	// 左臂电机
	axis_LeftArm_Wrist_MoveAbs									:MC_MoveAbsolute;			//左臂_腕电机MoveAbs功能块	
	axis_LeftArm_Left_MoveAbs									:MC_MoveAbsolute;			//左臂_左电机MoveAbs功能块
	axis_LeftArm_Right_MoveAbs									:MC_MoveAbsolute;			//左臂_右电机MoveAbs功能块
	axis_LeftArm_Lift_MoveAbs									:MC_MoveAbsolute;			//左臂_升电机MoveAbs功能块
	                                                                                                
	// 右臂电机                                                                                         
	axis_RightArm_Wrist_MoveAbs									:MC_MoveAbsolute;			//右臂_腕电机MoveAbs功能块	
	axis_RightArm_Left_MoveAbs									:MC_MoveAbsolute;			//右臂_左电机MoveAbs功能块
	axis_RightArm_Right_MoveAbs									:MC_MoveAbsolute;			//右臂_右电机MoveAbs功能块
	axis_RightArm_Lift_MoveAbs									:MC_MoveAbsolute;			//右臂_升电机MoveAbs功能块
	                                                                                               
	// 小龙门电机                                                                                        
	axis_SmallGate_Left_MoveAbs									:MC_MoveAbsolute;			//小门_左电机MoveAbs功能块
	axis_SmallGate_Right_MoveAbs								:MC_MoveAbsolute;			//小门_右电机MoveAbs功能块
	                                                                                               
	// 大龙门单电机                                                                                       
	axis_BigGate_Left_MoveAbs									:MC_MoveAbsolute;			//大门_左电机MoveAbs功能块
	axis_BigGate_Right_MoveAbs									:MC_MoveAbsolute;			//大门_右电机MoveAbs功能块
	                                                                                               
	// 后龙门单电机                                                                                      
	axis_BackGate_Left_MoveAbs									:MC_MoveAbsolute;			//后门_左电机MoveAbs功能块
	axis_BackGate_Right_MoveAbs									:MC_MoveAbsolute;			//后门_右电机MoveAbs功能块
	
	// 右轮
	axis_RightWheel_Steer_MoveAbs								:MC_MoveAbsolute;
	axis_RightWheel_Walk_MoveAbs								:MC_MoveAbsolute;
	
	// 左轮
	axis_LeftWheel_Steer_MoveAbs								:MC_MoveAbsolute;
	axis_LeftWheel_Walk_MoveAbs									:MC_MoveAbsolute;

(*======================================== 机器人各轴 MC_MoveAbs定义 End =====================================*)



(*====================================== 机器人各轴 MC_MoveVelocity定义 Start ================================*)

	axis_LeftWheel_Walk_MoveVelo								:MC_MoveVelocity;			// 左轮按速度运动
	axis_RightWheel_Walk_MoveVelo								:MC_MoveVelocity;			// 右轮按速度运动
	
(*====================================== 机器人各轴 MC_MoveVelocity定义 Stop ================================*)



(*======================================== 机器人各轴 MC_Stop定义 Start ==================================*)
	
	// 左臂电机
	axis_LeftArm_Wrist_McStop									:MC_Stop;			//左臂_腕电机MC_Stop块	
	axis_LeftArm_Left_McStop									:MC_Stop;			//左臂_左电机MC_Stop块
	axis_LeftArm_Right_McStop									:MC_Stop;			//左臂_右电机MC_Stop块
	axis_LeftArm_Lift_McStop									:MC_Stop;			//左臂_升电机MC_Stop块
	                                                                                        
	// 右臂电机                                                                                 
	axis_RightArm_Wrist_McStop									:MC_Stop;			//右臂_腕电机MC_Stop块	
	axis_RightArm_Left_McStop									:MC_Stop;			//右臂_左电机MC_Stop块
	axis_RightArm_Right_McStop									:MC_Stop;			//右臂_右电机MC_Stop块
	axis_RightArm_Lift_McStop									:MC_Stop;			//右臂_升电机MC_Stop块
	                                                                                        
	// 小龙门电机                                                                                
	axis_SmallGate_Left_McStop									:MC_Stop;			//小门_左电机MC_Stop块
	axis_SmallGate_Right_McStop									:MC_Stop;			//小门_右电机MC_Stop块
	                                                                                        
	// 大龙门单电机                                                                               
	axis_BigGate_Left_McStop									:MC_Stop;			//大门_左电机MC_Stop块
	axis_BigGate_Right_McStop									:MC_Stop;			//大门_右电机MC_Stop块
	                                                                                        
	// 后龙门单电机                                                                               
	axis_BackGate_Left_McStop									:MC_Stop;			//后门_左电机MC_Stop块
	axis_BackGate_Right_McStop									:MC_Stop;			//后门_右电机MC_Stop块

	// 右轮
	axis_RightWheel_Steer_McStop								:MC_Stop;;
	axis_RightWheel_Walk_McStop									:MC_Stop;
	
	// 左轮
	axis_LeftWheel_Steer_McStop									:MC_Stop;
	axis_LeftWheel_Walk_McStop									:MC_Stop;	
	

(*======================================== 机器人各轴 Mc_Stop定义 End =====================================*)




	

END_VAR

// ---- GVLs/Robot_Parameter.TcGVL
//{attribute 'qualified_only'}
VAR_GLOBAL
	
(* 测试臂参数
	
	//已知量
	h 						:LREAL:=260;
	i 						:LREAL:=260;
	g 						:LREAL:=150;
	f 						:LREAL:=150;
	w 						:LREAL:=110;
	angle_a					:LREAL:=137.5;			// 单位为度
	j						:LREAL:=40;
	n						:LREAL:=290.7497;     	// 余弦定理
	angle_FCE				:LREAL:=5.3330;			//余弦定理（单位为度）
*)

	// Left arm parameter
	LeftArm_h				:LREAL:=584.21;
	LeftArm_i				:LREAL:=500;
	LeftArm_g				:LREAL:=418;
	LeftArm_f				:LREAL:=418;
	LeftArm_w				:LREAL:=110;
	LeftArm_angle_a			:LREAL:=134.7;			//数模实测值,单位为度
	LeftArm_j				:LREAL:=147.73;
	LeftArm_n				:LREAL:=612.98;			//数模实测值
	LeftArm_angle_FCE		:LREAL:=9.86;			//数模实测值,单位为度
	
	// Right arm parameter
	RightArm_h				:LREAL:=500;
	RightArm_i				:LREAL:=584.21;
	RightArm_g				:LREAL:=418;
	RightArm_f				:LREAL:=418;
	RightArm_w				:LREAL:=110;
	RightArm_angle_a		:LREAL:=137.57;			//单位度
	RightArm_j				:LREAL:=147.73;
	RightArm_m				:LREAL:=617.76;
	RightArm_angle_FDE		:LREAL:=9.29;			//单位度

	//常量
	PI						:LREAL:=3.1415926;
	

END_VAR

// ---- GVLs/Robot_Status_Info.TcGVL
//{attribute 'qualified_only'}
VAR_GLOBAL
	
	(**********************************   电池相关参数    *************************************)
											
	Battery_TotalVoltage		AT%MW300		:LREAL;			 //voltage, unit: V
	Battery_TotalCurrent		AT%MW304		:LREAL;			 //current, unit:A
	Battery_RemainCapacity						:REAL;			 //remain capacitu, unit:Ah
	Battery_NominalCapacity						:REAL;			 //nominal capacity, unit:Ah
	Battery_CycleNum							:UINT;			 //cycle number, unit:times
	Battery_ProtectionMode						:WORD;			 //protection mode word
	Battery_RSOC								:USINT;			 //remain capacity, unit:%
	Battery_FETStatus							:BYTE;			 //mos fet status word
	Battery_humidity							:USINT;			 //humidity, unity:%
	Battery_WarningStatus						:WORD;			 //warning status word
	
	// 自定义标志位
	bBattery_Charging	   	 	    AT%MX10.0	:BOOL;			 //电池充放电状态标志位，电流正为充电，电流负为放电。
	bBattery_DisCharging		    AT%MX10.1	:BOOL;			 //电池充放电状态标志位，电流正为充电，电流负为放电。
	lrBattery_DisChargingCurrent	AT%MW304	:LREAL;			 //放电电流
	lrBattery_ChargingCurrent		AT%MW308	:LREAL;			 //充电电流
	lrBattery_RemainCapacity_Pecent AT%MW312	:LREAL;			 //剩余电量百分比，和Battery_RSOC不同，这个是用Battery_RemainCapacity、Battery_NominalCapacity两个参数算出来的。
	
	// Battery_ProtectionMode 电池保护状态定义标志位
	bSingleCellOvervoltageProtection    		: BOOL;			 // bit0: 单体过压保护
	bSingleCellUndervoltageProtection   		: BOOL;			 // bit1: 单体欠压保护
	bWholeGroupOvervoltageProtection    		: BOOL;			 // bit2: 整组过压保护
	bWholeGroupUndervoltageProtection   		: BOOL;			 // bit3: 整组欠压保护
	bChargingOverTemperatureProtection  		: BOOL;			 // bit4: 充电过温保护
	bChargingLowTemperatureProtection   		: BOOL;			 // bit5: 充电低温保护
	bDischargingOverTemperatureProtection		: BOOL;			 // bit6: 放电过温保护
	bDischargingLowTemperatureProtection		: BOOL;			 // bit7: 放电低温保护
	bChargingOvercurrentProtection      		: BOOL;			 // bit8: 充电过流保护
	bDischargingOvercurrentProtection   		: BOOL;			 // bit9: 放电过流保护
	bShortCircuitProtection             		: BOOL;			 // bit10: 短路保护
	bFrontEndDetectionICError           		: BOOL;			 // bit11: 前端检测IC错误
	bSoftwareLockedMOS                  		: BOOL;			 // bit12: 软件锁定MOS
	bChargingMOSBreakdownFlag           		: BOOL;			 // bit13: 充电MOS击穿标志
	bDischargingMOSBreakdownFlag        		: BOOL;			 // bit14: 放电MOS击穿标志
	bReserved                           		: BOOL;			 // bit15: 预留

	// Battery_FETStatus 电池MOS标志位
	bChargeMOSStatus    						: BOOL; 		// bit0: 充电MOS状态
	bDischargeMOSStatus 						: BOOL; 		// bit1: 放电MOS状态
	bCurrentLimitStatus 						: BOOL; 		// bit2: 限流模块状态
	bHeatingStatus      						: BOOL; 		// bit3: 加热模块状态
	
	// Battery Warning Status
	bSingleCellHighVoltageWarning    			: BOOL; 		// bit0: 单体高压告警
	bSingleCellLowVoltageWarning     			: BOOL; 		// bit1: 单体低压告警
	bWholeGroupHighVoltageWarning    			: BOOL; 		// bit2: 整组高压告警
	bWholeGroupLowVoltageWarning     			: BOOL; 		// bit3: 整组低压告警
	bChargingHighTemperatureWarning  			: BOOL; 		// bit4: 充电高温告警
	bChargingLowTemperatureWarning   			: BOOL; 		// bit5: 充电低温告警
	bDischargingHighTemperatureWarning			: BOOL; 		// bit6: 放电高温告警
	bDischargingLowTemperatureWarning 			: BOOL; 		// bit7: 放电低温保护
	bChargingHighCurrentWarning      			: BOOL; 		// bit8: 充电电流大告警
	bDischargingHighCurrentWarning   			: BOOL; 		// bit9: 放电电流大告警
	bSingleCellVoltageDifferenceWarning			: BOOL; 		// bit10: 单体压差大告警
	bLowCapacityWarning              			: BOOL; 		// bit11: 容量低告警
	bReserved12                      			: BOOL; 		// bit12: 预留
	bReserved13                      			: BOOL; 		// bit13: 预留
	bReserved14                      			: BOOL; 		// bit14: 预留
	
	
	



	(**********************************   轴相关参数    *************************************)
	
	// 伺服驱动器Error标志位
	bDriverDeviceError_axis_LeftArm_Left				AT%I*					:BOOL;		// 伺服驱动器报警_标志位_LeftArm_Left	
	bDriverDeviceError_axis_LeftArm_Right				AT%I*					:BOOL;		// 伺服驱动器报警_标志位_LeftArm_Right	
	bDriverDeviceError_axis_LeftArm_Wrist				AT%I*					:BOOL;		// 伺服驱动器报警_标志位_LeftArm_Wrist	
	bDriverDeviceError_axis_LeftArm_Lift				AT%I*					:BOOL;		// 伺服驱动器报警_标志位_LeftArm_Lift	
	bDriverDeviceError_axis_RightArm_Left				AT%I*					:BOOL;		// 伺服驱动器报警_标志位_RightArm_Left	
	bDriverDeviceError_axis_RightArm_Right				AT%I*					:BOOL;      // 伺服驱动器报警_标志位_RightArm_Right	
	bDriverDeviceError_axis_RightArm_Wrist				AT%I*					:BOOL;      // 伺服驱动器报警_标志位_RightArm_Wrist	
	bDriverDeviceError_axis_RightArm_Lift				AT%I*					:BOOL;	    // 伺服驱动器报警_标志位_RightArm_Lift	
	bDriverDeviceError_axis_BigGate_Left				AT%I*					:BOOL;		// 伺服驱动器报警_标志位_BigGate_Left
	bDriverDeviceError_axis_BigGate_Right				AT%I*					:BOOL;      // 伺服驱动器报警_标志位_BigGate_Right
	bDriverDeviceError_axis_SmallGate_Left				AT%I*					:BOOL;      // 伺服驱动器报警_标志位_SmallGate_Left
	bDriverDeviceError_axis_SmallGate_Right				AT%I*					:BOOL;      // 伺服驱动器报警_标志位_SmallGate_Right
	bDriverDeviceError_axis_BackGate_Left				AT%I*					:BOOL;		// 伺服驱动器报警_标志位_BackGate_Left
	bDriverDeviceError_axis_BackGate_Right				AT%I*					:BOOL;	    // 伺服驱动器报警_标志位_BackGate_Right
	bDriverDeviceError_axis_RightWheel_Steer			AT%I*					:BOOL;      // 伺服驱动器报警_标志位_RightWheel_Steer
	bDriverDeviceError_axis_RightWheel_Walk				AT%I*					:BOOL;		// 伺服驱动器报警_标志位_RightWheel_Walk
	bDriverDeviceError_axis_LeftWheel_Steer				AT%I*					:BOOL;		// 伺服驱动器报警_标志位_LeftWheel_Steer
	bDriverDeviceError_axis_LeftWheel_Walk				AT%I*					:BOOL;		// 伺服驱动器报警_标志位_LeftWheel_Walk
	
	// 伺服驱动器ErrorCode
	bDriverDeviceErrorCode_axis_LeftArm_Left			AT%I*					:UDINT;		// 伺服驱动器报警_错误代码_LeftArm_Left	
	bDriverDeviceErrorCode_axis_LeftArm_Right			AT%I*					:UDINT;		// 伺服驱动器报警_错误代码_LeftArm_Right	
	bDriverDeviceErrorCode_axis_LeftArm_Wrist			AT%I*					:UDINT;		// 伺服驱动器报警_错误代码_LeftArm_Wrist	
	bDriverDeviceErrorCode_axis_LeftArm_Lift			AT%I*					:UDINT;		// 伺服驱动器报警_错误代码_LeftArm_Lift	
	bDriverDeviceErrorCode_axis_RightArm_Left			AT%I*					:UDINT;		// 伺服驱动器报警_错误代码_RightArm_Left	
	bDriverDeviceErrorCode_axis_RightArm_Right			AT%I*					:UDINT;      // 伺服驱动器报警_错误代码_RightArm_Right	
	bDriverDeviceErrorCode_axis_RightArm_Wrist			AT%I*					:UDINT;      // 伺服驱动器报警_错误代码_RightArm_Wrist	
	bDriverDeviceErrorCode_axis_RightArm_Lift			AT%I*					:UDINT;	    // 伺服驱动器报警_错误代码_RightArm_Lift	
	bDriverDeviceErrorCode_axis_BigGate_Left			AT%I*					:UDINT;		// 伺服驱动器报警_错误代码_BigGate_Left
	bDriverDeviceErrorCode_axis_BigGate_Right			AT%I*					:UDINT;      // 伺服驱动器报警_错误代码_BigGate_Right
	bDriverDeviceErrorCode_axis_SmallGate_Left			AT%I*					:UDINT;      // 伺服驱动器报警_错误代码_SmallGate_Left
	bDriverDeviceErrorCode_axis_SmallGate_Right			AT%I*					:UDINT;      // 伺服驱动器报警_错误代码_SmallGate_Right
	bDriverDeviceErrorCode_axis_BackGate_Left			AT%I*					:UDINT;		// 伺服驱动器报警_错误代码_BackGate_Left
	bDriverDeviceErrorCode_axis_BackGate_Right			AT%I*					:UDINT;	    // 伺服驱动器报警_错误代码_BackGate_Right
	bDriverDeviceErrorCode_axis_RightWheel_Steer		AT%I*					:UDINT;      // 伺服驱动器报警_错误代码_RightWheel_Steer
	bDriverDeviceErrorCode_axis_RightWheel_Walk			AT%I*					:UDINT;		// 伺服驱动器报警_错误代码_RightWheel_Walk
	bDriverDeviceErrorCode_axis_LeftWheel_Steer			AT%I*					:UDINT;		// 伺服驱动器报警_错误代码_LeftWheel_Steer
	bDriverDeviceErrorCode_axis_LeftWheel_Walk			AT%I*					:UDINT;		// 伺服驱动器报警_错误代码_LeftWheel_Walk
	
END_VAR

// ---- POUs/AxisAbs.TcPOU
PROGRAM AxisAbs
VAR
	nSpeed_MoveAbs						:LREAL:=5;
	
	nTargetPos_MoveAbs								:LREAL;

END_VAR


// LeftArm_Left_MoveAbs
IF bManualCtrl_Part_LeftArm_Left THEN					
	axis_LeftArm_Left_MoveAbs(
		Axis:= axis_LeftArm_Left, 
		Execute:= bAxis_LeftArm_Left_MoveAbs, 
		Position:= nTargetPos_MoveAbs, 
		Velocity:= nSpeed_MoveAbs, 
		Acceleration:= , 
		Deceleration:= , 
		Jerk:= , 
		BufferMode:= , 
		Options:= , 
		Done=> , 
		Busy=> , 
		Active=> , 
		CommandAborted=> , 
		Error=> , 
		ErrorID=> );	
END_IF

// LeftArm_Right_MoveAbs
IF bManualCtrl_Part_LeftArm_Right THEN					
	axis_LeftArm_Right_MoveAbs(
		Axis:= axis_LeftArm_Right, 
		Execute:= bAxis_LeftArm_Right_MoveAbs, 
		Position:= nTargetPos_MoveAbs, 
		Velocity:= nSpeed_MoveAbs, 
		Acceleration:= , 
		Deceleration:= , 
		Jerk:= , 
		BufferMode:= , 
		Options:= , 
		Done=> , 
		Busy=> , 
		Active=> , 
		CommandAborted=> , 
		Error=> , 
		ErrorID=> );	
END_IF


// LeftArm_Wrist_MoveAbs
IF bManualCtrl_Part_LeftArm_Wrist THEN					
	axis_LeftArm_Wrist_MoveAbs(
		Axis:= axis_LeftArm_Wrist, 
		Execute:= bAxis_LeftArm_Wrist_MoveAbs, 
		Position:= nTargetPos_MoveAbs, 
		Velocity:= nSpeed_MoveAbs, 
		Acceleration:= , 
		Deceleration:= , 
		Jerk:= , 
		BufferMode:= , 
		Options:= , 
		Done=> , 
		Busy=> , 
		Active=> , 
		CommandAborted=> , 
		Error=> , 
		ErrorID=> );	
END_IF


// LeftArm_Lift_MoveAbs
IF bManualCtrl_Part_LeftArm_Lift THEN					
	axis_LeftArm_Lift_MoveAbs(
		Axis:= axis_LeftArm_Lift, 
		Execute:= bAxis_LeftArm_Lift_MoveAbs, 
		Position:= nTargetPos_MoveAbs, 
		Velocity:= nSpeed_MoveAbs, 
		Acceleration:= , 
		Deceleration:= , 
		Jerk:= , 
		BufferMode:= , 
		Options:= , 
		Done=> , 
		Busy=> , 
		Active=> , 
		CommandAborted=> , 
		Error=> , 
		ErrorID=> );	
END_IF



// RightArm_Left_MoveAbs
IF bManualCtrl_Part_RightArm_Left THEN					
	axis_RightArm_Left_MoveAbs(
		Axis:= axis_RightArm_Left, 
		Execute:= bAxis_RightArm_Left_MoveAbs, 
		Position:= nTargetPos_MoveAbs, 
		Velocity:= nSpeed_MoveAbs, 
		Acceleration:= , 
		Deceleration:= , 
		Jerk:= , 
		BufferMode:= , 
		Options:= , 
		Done=> , 
		Busy=> , 
		Active=> , 
		CommandAborted=> , 
		Error=> , 
		ErrorID=> );	
END_IF

// RightArm_Right_MoveAbs
IF bManualCtrl_Part_RightArm_Right THEN					
	axis_RightArm_Right_MoveAbs(
		Axis:= axis_RightArm_Right, 
		Execute:= bAxis_RightArm_Right_MoveAbs, 
		Position:= nTargetPos_MoveAbs, 
		Velocity:= nSpeed_MoveAbs, 
		Acceleration:= , 
		Deceleration:= , 
		Jerk:= , 
		BufferMode:= , 
		Options:= , 
		Done=> , 
		Busy=> , 
		Active=> , 
		CommandAborted=> , 
		Error=> , 
		ErrorID=> );	
END_IF


// RightArm_Wrist_MoveAbs
IF bManualCtrl_Part_RightArm_Wrist THEN					
	axis_RightArm_Wrist_MoveAbs(
		Axis:= axis_RightArm_Wrist, 
		Execute:= bAxis_RightArm_Wrist_MoveAbs, 
		Position:= nTargetPos_MoveAbs, 
		Velocity:= nSpeed_MoveAbs, 
		Acceleration:= , 
		Deceleration:= , 
		Jerk:= , 
		BufferMode:= , 
		Options:= , 
		Done=> , 
		Busy=> , 
		Active=> , 
		CommandAborted=> , 
		Error=> , 
		ErrorID=> );	
END_IF


// RightArm_Lift_MoveAbs
IF bManualCtrl_Part_RightArm_Lift THEN					
	axis_RightArm_Lift_MoveAbs(
		Axis:= axis_RightArm_Lift, 
		Execute:= bAxis_RightArm_Lift_MoveAbs, 
		Position:= nTargetPos_MoveAbs, 
		Velocity:= nSpeed_MoveAbs, 
		Acceleration:= , 
		Deceleration:= , 
		Jerk:= , 
		BufferMode:= , 
		Options:= , 
		Done=> , 
		Busy=> , 
		Active=> , 
		CommandAborted=> , 
		Error=> , 
		ErrorID=> );	
END_IF


// BigGate_Left_MoveAbs
IF bManualCtrl_Part_BigGate_Left THEN					
	axis_BigGate_Left_MoveAbs(
		Axis:= axis_BigGate_Left, 
		Execute:= bAxis_BigGate_Left_MoveAbs, 
		Position:= nTargetPos_MoveAbs, 
		Velocity:= nSpeed_MoveAbs, 
		Acceleration:= , 
		Deceleration:= , 
		Jerk:= , 
		BufferMode:= , 
		Options:= , 
		Done=> , 
		Busy=> , 
		Active=> , 
		CommandAborted=> , 
		Error=> , 
		ErrorID=> );	
END_IF

// BigGate_Right_MoveAbs
IF bManualCtrl_Part_BigGate_Right THEN					
	axis_BigGate_Right_MoveAbs(
		Axis:= axis_BigGate_Right, 
		Execute:= bAxis_BigGate_Right_MoveAbs, 
		Position:= nTargetPos_MoveAbs, 
		Velocity:= nSpeed_MoveAbs, 
		Acceleration:= , 
		Deceleration:= , 
		Jerk:= , 
		BufferMode:= , 
		Options:= , 
		Done=> , 
		Busy=> , 
		Active=> , 
		CommandAborted=> , 
		Error=> , 
		ErrorID=> );	
END_IF

// SmallGate_Left_MoveAbs
IF bManualCtrl_Part_SmallGate_Left THEN					
	axis_SmallGate_Left_MoveAbs(
		Axis:= axis_SmallGate_Left, 
		Execute:= bAxis_SmallGate_Left_MoveAbs, 
		Position:= nTargetPos_MoveAbs, 
		Velocity:= nSpeed_MoveAbs, 
		Acceleration:= , 
		Deceleration:= , 
		Jerk:= , 
		BufferMode:= , 
		Options:= , 
		Done=> , 
		Busy=> , 
		Active=> , 
		CommandAborted=> , 
		Error=> , 
		ErrorID=> );	
END_IF

// SmallGate_Right_MoveAbs
IF bManualCtrl_Part_SmallGate_Right THEN					
	axis_SmallGate_Right_MoveAbs(
		Axis:= axis_SmallGate_Right, 
		Execute:= bAxis_SmallGate_Right_MoveAbs, 
		Position:= nTargetPos_MoveAbs, 
		Velocity:= nSpeed_MoveAbs, 
		Acceleration:= , 
		Deceleration:= , 
		Jerk:= , 
		BufferMode:= , 
		Options:= , 
		Done=> , 
		Busy=> , 
		Active=> , 
		CommandAborted=> , 
		Error=> , 
		ErrorID=> );	
END_IF


// BackGate_Left_MoveAbs
IF bManualCtrl_Part_BackGate_Left THEN					
	axis_BackGate_Left_MoveAbs(
		Axis:= axis_BackGate_Left, 
		Execute:= bAxis_BackGate_Left_MoveAbs, 
		Position:= nTargetPos_MoveAbs, 
		Velocity:= nSpeed_MoveAbs, 
		Acceleration:= , 
		Deceleration:= , 
		Jerk:= , 
		BufferMode:= , 
		Options:= , 
		Done=> , 
		Busy=> , 
		Active=> , 
		CommandAborted=> , 
		Error=> , 
		ErrorID=> );	
END_IF

// BackGate_Right_MoveAbs
IF bManualCtrl_Part_BackGate_Right THEN					
	axis_BackGate_Right_MoveAbs(
		Axis:= axis_BackGate_Right, 
		Execute:= bAxis_BackGate_Right_MoveAbs, 
		Position:= nTargetPos_MoveAbs, 
		Velocity:= nSpeed_MoveAbs, 
		Acceleration:= , 
		Deceleration:= , 
		Jerk:= , 
		BufferMode:= , 
		Options:= , 
		Done=> , 
		Busy=> , 
		Active=> , 
		CommandAborted=> , 
		Error=> , 
		ErrorID=> );	
END_IF

END_PROGRAM

// ---- POUs/AxisAllCtrl.TcPOU
PROGRAM AxisAllCtrl
VAR
	i				:USINT := 1;

END_VAR



//所有Axis上电
IF bAxis_All_Enable THEN
	FOR i:=1 TO nAxisNum DO
		aAxis_All_Enable_Group[i]^:=TRUE;
	END_FOR
END_IF

//所有Axis下电
IF bAxis_All_Disable THEN
	FOR i:=1 TO nAxisNum DO
		aAxis_All_Enable_Group[i]^:=FALSE;
	END_FOR
END_IF

//所有轴清除故障
IF bAxis_All_Reset THEN
	FOR i:=1 TO nAxisNum DO
		aAxis_All_Reset_Group[i]^:=TRUE;
	END_FOR
ELSE
	FOR i:=1 TO nAxisNum DO
		aAxis_All_Reset_Group[i]^:=FALSE;
	END_FOR	
END_IF

END_PROGRAM

// ---- POUs/AxisJog.TcPOU
PROGRAM AxisJog
VAR
	lrJogSpeed	: POINTER TO LREAL;
END_VAR

// 快速Jog速度设定
IF bJogFast THEN
	lrJogSpeed := ADR(aAxis_Jog_Speed[1]);
ELSE
	lrJogSpeed := ADR(aAxis_Jog_Speed[0]);
END_IF

// LeftArm_Left_Jog
IF bManualCtrl_Part_LeftArm_Left THEN

	axis_LeftArm_Left_Jog(
		Axis:= axis_LeftArm_Left, 
		JogForward:= bAxis_LeftArm_Left_JogP , 			// 如果想ABS的时候按下JOG按键不停止ABS动作就加上后面的判断AND NOT axis_LeftArm_Left_MoveAbs.Active
		JogBackwards:= bAxis_LeftArm_Left_JogN, 		// 如果想ABS的时候按下JOG按键不停止ABS动作就加上后面的判断AND NOT axis_LeftArm_Left_MoveAbs.Active
		Mode:= MC_JOGMODE_CONTINOUS, 					//需要设置为MC_JOGMODE_CONTINOUS下面的速度设定才有效
		Position:= , 
		Velocity:= lrJogSpeed^, 
		Acceleration:= , 
		Deceleration:= , 
		Jerk:= , 
		Done=> , 
		Busy=> , 
		Active=> , 
		CommandAborted=> , 
		Error=> , 
		ErrorID=> );

END_IF

// LeftArm_Right_Jog
IF bManualCtrl_Part_LeftArm_Right THEN

	axis_LeftArm_Right_Jog(
		Axis:= axis_LeftArm_Right, 
		JogForward:= bAxis_LeftArm_Right_JogP , 			
		JogBackwards:= bAxis_LeftArm_Right_JogN, 		
		Mode:= MC_JOGMODE_CONTINOUS, 					//需要设置为MC_JOGMODE_CONTINOUS下面的速度设定才有效
		Position:= , 
		Velocity:= lrJogSpeed^, 
		Acceleration:= , 
		Deceleration:= , 
		Jerk:= , 
		Done=> , 
		Busy=> , 
		Active=> , 
		CommandAborted=> , 
		Error=> , 
		ErrorID=> );

END_IF

// LeftArm_Wrist_Jog
IF bManualCtrl_Part_LeftArm_Wrist THEN

	axis_LeftArm_Right_Jog(
		Axis:= axis_LeftArm_Wrist, 
		JogForward:= bAxis_LeftArm_Wrist_JogP , 			
		JogBackwards:= bAxis_LeftArm_Wrist_JogN, 		
		Mode:= MC_JOGMODE_CONTINOUS, 					//需要设置为MC_JOGMODE_CONTINOUS下面的速度设定才有效
		Position:= , 
		Velocity:= lrJogSpeed^, 
		Acceleration:= , 
		Deceleration:= , 
		Jerk:= , 
		Done=> , 
		Busy=> , 
		Active=> , 
		CommandAborted=> , 
		Error=> , 
		ErrorID=> );

END_IF


// LeftArm_Lift_Jog
IF bManualCtrl_Part_LeftArm_Lift THEN

	axis_LeftArm_Lift_Jog(
		Axis:= axis_LeftArm_Lift, 
		JogForward:= bAxis_LeftArm_Lift_JogP , 			
		JogBackwards:= bAxis_LeftArm_Lift_JogN, 		
		Mode:= MC_JOGMODE_CONTINOUS, 					//需要设置为MC_JOGMODE_CONTINOUS下面的速度设定才有效
		Position:= , 
		Velocity:= lrJogSpeed^, 
		Acceleration:= , 
		Deceleration:= , 
		Jerk:= , 
		Done=> , 
		Busy=> , 
		Active=> , 
		CommandAborted=> , 
		Error=> , 
		ErrorID=> );

END_IF



// RightArm_Left_Jog
IF bManualCtrl_Part_RightArm_Left THEN

	axis_RightArm_Left_Jog(
		Axis:= axis_RightArm_Left, 
		JogForward:= bAxis_RightArm_Left_JogP , 			// 如果想ABS的时候按下JOG按键不停止ABS动作就加上后面的判断AND NOT axis_LeftArm_Left_MoveAbs.Active
		JogBackwards:= bAxis_RightArm_Left_JogN, 		// 如果想ABS的时候按下JOG按键不停止ABS动作就加上后面的判断AND NOT axis_LeftArm_Left_MoveAbs.Active
		Mode:= MC_JOGMODE_CONTINOUS, 					//需要设置为MC_JOGMODE_CONTINOUS下面的速度设定才有效
		Position:= , 
		Velocity:= lrJogSpeed^, 
		Acceleration:= , 
		Deceleration:= , 
		Jerk:= , 
		Done=> , 
		Busy=> , 
		Active=> , 
		CommandAborted=> , 
		Error=> , 
		ErrorID=> );

END_IF

// RightArm_Right_Jog
IF bManualCtrl_Part_RightArm_Right THEN

	axis_RightArm_Right_Jog(
		Axis:= axis_RightArm_Right, 
		JogForward:= bAxis_RightArm_Right_JogP , 			
		JogBackwards:= bAxis_RightArm_Right_JogN, 		
		Mode:= MC_JOGMODE_CONTINOUS, 					//需要设置为MC_JOGMODE_CONTINOUS下面的速度设定才有效
		Position:= , 
		Velocity:= lrJogSpeed^, 
		Acceleration:= , 
		Deceleration:= , 
		Jerk:= , 
		Done=> , 
		Busy=> , 
		Active=> , 
		CommandAborted=> , 
		Error=> , 
		ErrorID=> );

END_IF

// RightArm_Wrist_Jog
IF bManualCtrl_Part_RightArm_Wrist THEN

	axis_RightArm_Right_Jog(
		Axis:= axis_RightArm_Wrist, 
		JogForward:= bAxis_RightArm_Wrist_JogP , 			
		JogBackwards:= bAxis_RightArm_Wrist_JogN, 		
		Mode:= MC_JOGMODE_CONTINOUS, 					//需要设置为MC_JOGMODE_CONTINOUS下面的速度设定才有效
		Position:= , 
		Velocity:= lrJogSpeed^, 
		Acceleration:= , 
		Deceleration:= , 
		Jerk:= , 
		Done=> , 
		Busy=> , 
		Active=> , 
		CommandAborted=> , 
		Error=> , 
		ErrorID=> );

END_IF


// RightArm_Lift_Jog
IF bManualCtrl_Part_RightArm_Lift THEN

	axis_RightArm_Lift_Jog(
		Axis:= axis_RightArm_Lift, 
		JogForward:= bAxis_RightArm_Lift_JogP , 			
		JogBackwards:= bAxis_RightArm_Lift_JogN, 		
		Mode:= MC_JOGMODE_CONTINOUS, 					//需要设置为MC_JOGMODE_CONTINOUS下面的速度设定才有效
		Position:= , 
		Velocity:= lrJogSpeed^, 
		Acceleration:= , 
		Deceleration:= , 
		Jerk:= , 
		Done=> , 
		Busy=> , 
		Active=> , 
		CommandAborted=> , 
		Error=> , 
		ErrorID=> );

END_IF


// BigGate_Left_Jog(正转升，反转降)
IF bManualCtrl_Part_BigGate_Left THEN

	axis_BigGate_Left_Jog(
		Axis:= axis_BigGate_Left, 
		JogForward:= bAxis_BigGate_Left_JogP , 			// 如果想ABS的时候按下JOG按键不停止ABS动作就加上后面的判断AND NOT axis_LeftArm_Left_MoveAbs.Active
		JogBackwards:= bAxis_BigGate_Left_JogN, 		// 如果想ABS的时候按下JOG按键不停止ABS动作就加上后面的判断AND NOT axis_LeftArm_Left_MoveAbs.Active
		Mode:= MC_JOGMODE_CONTINOUS, 					//需要设置为MC_JOGMODE_CONTINOUS下面的速度设定才有效
		Position:= , 
		Velocity:= lrJogSpeed^, 
		Acceleration:= , 
		Deceleration:= , 
		Jerk:= , 
		Done=> , 
		Busy=> , 
		Active=> , 
		CommandAborted=> , 
		Error=> , 
		ErrorID=> );

END_IF

// BigGate_Right_Jog(正转降反转升)
IF bManualCtrl_Part_BigGate_Right THEN

	axis_BigGate_Right_Jog(
		Axis:= axis_BigGate_Right, 
		JogForward:= bAxis_BigGate_Right_JogP , 			
		JogBackwards:= bAxis_BigGate_Right_JogN, 		
		Mode:= MC_JOGMODE_CONTINOUS, 					//需要设置为MC_JOGMODE_CONTINOUS下面的速度设定才有效
		Position:= , 
		Velocity:= lrJogSpeed^, 
		Acceleration:= , 
		Deceleration:= , 
		Jerk:= , 
		Done=> , 
		Busy=> , 
		Active=> , 
		CommandAborted=> , 
		Error=> , 
		ErrorID=> );

END_IF


// SmallGate_Left_Jog
IF bManualCtrl_Part_SmallGate_Left THEN

	axis_SmallGate_Left_Jog(
		Axis:= axis_SmallGate_Left, 
		JogForward:= bAxis_SmallGate_Left_JogP , 			// 如果想ABS的时候按下JOG按键不停止ABS动作就加上后面的判断AND NOT axis_LeftArm_Left_MoveAbs.Active
		JogBackwards:= bAxis_SmallGate_Left_JogN, 		// 如果想ABS的时候按下JOG按键不停止ABS动作就加上后面的判断AND NOT axis_LeftArm_Left_MoveAbs.Active
		Mode:= MC_JOGMODE_CONTINOUS, 					//需要设置为MC_JOGMODE_CONTINOUS下面的速度设定才有效
		Position:= , 
		Velocity:= lrJogSpeed^, 
		Acceleration:= , 
		Deceleration:= , 
		Jerk:= , 
		Done=> , 
		Busy=> , 
		Active=> , 
		CommandAborted=> , 
		Error=> , 
		ErrorID=> );

END_IF

// SmallGate_Right_Jog
IF bManualCtrl_Part_SmallGate_Right THEN

	axis_SmallGate_Right_Jog(
		Axis:= axis_SmallGate_Right, 
		JogForward:= bAxis_SmallGate_Right_JogP , 			
		JogBackwards:= bAxis_SmallGate_Right_JogN, 		
		Mode:= MC_JOGMODE_CONTINOUS, 					//需要设置为MC_JOGMODE_CONTINOUS下面的速度设定才有效
		Position:= , 
		Velocity:= lrJogSpeed^, 
		Acceleration:= , 
		Deceleration:= , 
		Jerk:= , 
		Done=> , 
		Busy=> , 
		Active=> , 
		CommandAborted=> , 
		Error=> , 
		ErrorID=> );

END_IF



// BackGate_Left_Jog
IF bManualCtrl_Part_BackGate_Left THEN

	axis_BackGate_Left_Jog(
		Axis:= axis_BackGate_Left, 
		JogForward:= bAxis_BackGate_Left_JogP , 			// 如果想ABS的时候按下JOG按键不停止ABS动作就加上后面的判断AND NOT axis_LeftArm_Left_MoveAbs.Active
		JogBackwards:= bAxis_BackGate_Left_JogN, 		// 如果想ABS的时候按下JOG按键不停止ABS动作就加上后面的判断AND NOT axis_LeftArm_Left_MoveAbs.Active
		Mode:= MC_JOGMODE_CONTINOUS, 					//需要设置为MC_JOGMODE_CONTINOUS下面的速度设定才有效
		Position:= , 
		Velocity:= lrJogSpeed^, 
		Acceleration:= , 
		Deceleration:= , 
		Jerk:= , 
		Done=> , 
		Busy=> , 
		Active=> , 
		CommandAborted=> , 
		Error=> , 
		ErrorID=> );

END_IF

// BackGate_Right_Jog
IF bManualCtrl_Part_BackGate_Right THEN

	axis_BackGate_Right_Jog(
		Axis:= axis_BackGate_Right, 
		JogForward:= bAxis_BackGate_Right_JogP , 			
		JogBackwards:= bAxis_BackGate_Right_JogN, 		
		Mode:= MC_JOGMODE_CONTINOUS, 					//需要设置为MC_JOGMODE_CONTINOUS下面的速度设定才有效
		Position:= , 
		Velocity:= lrJogSpeed^, 
		Acceleration:= , 
		Deceleration:= , 
		Jerk:= , 
		Done=> , 
		Busy=> , 
		Active=> , 
		CommandAborted=> , 
		Error=> , 
		ErrorID=> );

END_IF

END_PROGRAM

// ---- POUs/AxisPowerOn.TcPOU
PROGRAM AxisPowerOn
VAR

END_VAR


//左臂-左电机-PowerOn
axis_LeftArm_Left_Power(
	Axis:= axis_LeftArm_Left, 
	Enable:= bAxis_LeftArm_Left_Enable, 
	Enable_Positive:= TRUE, 
	Enable_Negative:= TRUE, 
	Override:= , 
	BufferMode:= , 
	Options:= , 
	Status=> axis_LeftArm_Left_Power_Output.Done, 
	Busy=> , 
	Error=> , 
	ErrorID=> );
	
	
//左臂-右电机-PowerOn
axis_LeftArm_Right_Power(
	Axis:= axis_LeftArm_Right, 
	Enable:= bAxis_LeftArm_Right_Enable, 
	Enable_Positive:= TRUE, 
	Enable_Negative:= TRUE, 
	Override:= , 
	BufferMode:= , 
	Options:= , 
	Status=> axis_LeftArm_Right_Power_Output.Done, 
	Busy=> , 
	Error=> , 
	ErrorID=> );
	
axis_LeftArm_Lift_Power(
	Axis:= axis_LeftArm_Lift, 
	Enable:= bAxis_LeftArm_Lift_Enable, 
	Enable_Positive:= TRUE, 
	Enable_Negative:= TRUE, 
	Override:= , 
	BufferMode:= , 
	Options:= , 
	Status=> , 
	Busy=> , 
	Error=> , 
	ErrorID=> );

axis_LeftArm_Wrist_Power(
	Axis:= axis_LeftArm_Wrist, 
	Enable:= bAxis_LeftArm_Wrist_Enable, 
	Enable_Positive:= TRUE, 
	Enable_Negative:= TRUE, 
	Override:= , 
	BufferMode:= , 
	Options:= , 
	Status=> , 
	Busy=> , 
	Error=> , 
	ErrorID=> );




//右臂-左电机-PowerOn
axis_RightArm_Left_Power(
	Axis:= axis_RightArm_Left, 
	Enable:= bAxis_RightArm_Left_Enable, 
	Enable_Positive:= TRUE, 
	Enable_Negative:= TRUE, 
	Override:= , 
	BufferMode:= , 
	Options:= , 
	Status=> axis_RightArm_Left_Power_Output.Done, 
	Busy=> , 
	Error=> , 
	ErrorID=> );
	
	
//右臂-右电机-PowerOn
axis_RightArm_Right_Power(
	Axis:= axis_RightArm_Right, 
	Enable:= bAxis_RightArm_Right_Enable, 
	Enable_Positive:= TRUE, 
	Enable_Negative:= TRUE, 
	Override:= , 
	BufferMode:= , 
	Options:= , 
	Status=> axis_RightArm_Right_Power_Output.Done, 
	Busy=> , 
	Error=> , 
	ErrorID=> );

//右臂-升电机-Poweron
axis_RightArm_Lift_Power(
	Axis:= axis_RightArm_Lift, 
	Enable:= bAxis_RightArm_Lift_Enable, 
	Enable_Positive:= TRUE, 
	Enable_Negative:= TRUE, 
	Override:= , 
	BufferMode:= , 
	Options:= , 
	Status=> , 
	Busy=> , 
	Error=> , 
	ErrorID=> );

//右臂-腕电机-Poweron
axis_RightArm_Wrist_Power(
	Axis:= axis_RightArm_Wrist, 
	Enable:= bAxis_RightArm_Wrist_Enable, 
	Enable_Positive:= TRUE, 
	Enable_Negative:= TRUE, 
	Override:= , 
	BufferMode:= , 
	Options:= , 
	Status=> axis_RightArm_Wrist_Power_Output.Done, 
	Busy=> , 
	Error=> , 
	ErrorID=> );
	


	
//大龙门-左电机-上电
axis_BigGate_Left_Power(
	Axis:= axis_BigGate_Left, 
	Enable:= bAxis_BigGate_Left_Enable, 
	Enable_Positive:= TRUE, 
	Enable_Negative:= TRUE, 
	Override:= , 
	BufferMode:= , 
	Options:= , 
	Status=> axis_BigGate_Left_Power_Output.Done, 
	Busy=> , 
	Error=> , 
	ErrorID=> );
	
//大龙门-右电机-上电	
axis_BigGate_Right_Power(
	Axis:= axis_BigGate_Right, 
	Enable:= bAxis_BigGate_Right_Enable, 
	Enable_Positive:= TRUE, 
	Enable_Negative:= TRUE, 
	Override:= , 
	BufferMode:= , 
	Options:= , 
	Status=> axis_BigGate_Right_Power_Output.Done, 
	Busy=> , 
	Error=> , 
	ErrorID=> );

//小龙门-左电机-上电	
axis_SmallGate_Left_Power(
	Axis:= axis_SmallGate_Left, 
	Enable:= bAxis_SmallGate_Left_Enable, 
	Enable_Positive:= TRUE, 
	Enable_Negative:= TRUE, 
	Override:= , 
	BufferMode:= , 
	Options:= , 
	Status=> axis_SmallGate_Left_Power_Output.Done, 
	Busy=> , 
	Error=> , 
	ErrorID=> );
	
//小龙门-右电机-上电	
axis_SmallGate_Right_Power(
	Axis:= axis_SmallGate_Right, 
	Enable:= bAxis_SmallGate_Right_Enable, 
	Enable_Positive:= TRUE, 
	Enable_Negative:= TRUE, 
	Override:= , 
	BufferMode:= , 
	Options:= , 
	Status=> axis_SmallGate_Right_Power_Output.Done, 
	Busy=> , 
	Error=> , 
	ErrorID=> );

//后龙门-左电机-上电	
axis_BackGate_Left_Power(
	Axis:= axis_BackGate_Left, 
	Enable:= bAxis_BackGate_Left_Enable, 
	Enable_Positive:= TRUE, 
	Enable_Negative:= TRUE, 
	Override:= , 
	BufferMode:= , 
	Options:= , 
	Status=> axis_BackGate_Left_Power_Output.Done, 
	Busy=> , 
	Error=> , 
	ErrorID=> );

//后龙门-右电机-上电
axis_BackGate_Right_Power(
	Axis:= axis_BackGate_Right, 
	Enable:= bAxis_BackGate_Right_Enable, 
	Enable_Positive:= TRUE, 
	Enable_Negative:= TRUE, 
	Override:= , 
	BufferMode:= , 
	Options:= , 
	Status=> axis_BackGate_Right_Power_Output.Done, 
	Busy=> , 
	Error=> , 
	ErrorID=> );

END_PROGRAM

// ---- POUs/AxisReset.TcPOU
PROGRAM AxisReset
VAR
END_VAR

//左臂
axis_LeftArm_Left_Reset(
	Axis:= axis_LeftArm_Left, 
	Execute:= bAxis_LeftArm_Left_Reset, 
	Done=> , 
	Busy=> , 
	Error=> , 
	ErrorID=> );
	
axis_LeftArm_Right_Reset(
	Axis:= axis_LeftArm_Right, 
	Execute:= bAxis_LeftArm_Right_Reset, 
	Done=> , 
	Busy=> , 
	Error=> , 
	ErrorID=> );

axis_LeftArm_Lift_Reset(
	Axis:= axis_LeftArm_Lift, 
	Execute:= bAxis_LeftArm_Lift_Reset, 
	Done=> , 
	Busy=> , 
	Error=> , 
	ErrorID=> );

axis_LeftArm_Wrist_Reset(
	Axis:= axis_LeftArm_Wrist, 
	Execute:= bAxis_LeftArm_Wrist_Reset, 
	Done=> , 
	Busy=> , 
	Error=> , 
	ErrorID=> );
	

//右臂
axis_RightArm_Left_Reset(
	Axis:= axis_RightArm_Left, 
	Execute:= bAxis_RightArm_Left_Reset, 
	Done=> , 
	Busy=> , 
	Error=> , 
	ErrorID=> );
	
axis_RightArm_Right_Reset(
	Axis:= axis_RightArm_Right, 
	Execute:= bAxis_RightArm_Right_Reset, 
	Done=> , 
	Busy=> , 
	Error=> , 
	ErrorID=> );

axis_RightArm_Lift_Reset(
	Axis:= axis_RightArm_Lift, 
	Execute:= bAxis_RightArm_Lift_Reset, 
	Done=> , 
	Busy=> , 
	Error=> , 
	ErrorID=> );

axis_RightArm_Wrist_Reset(
	Axis:= axis_RightArm_Wrist, 
	Execute:= bAxis_RightArm_Wrist_Reset, 
	Done=> , 
	Busy=> , 
	Error=> , 
	ErrorID=> );

//大龙门
axis_BigGate_Left_Reset(
	Axis:= axis_BigGate_Left, 
	Execute:= bAxis_BigGate_Left_Reset, 
	Done=> , 
	Busy=> , 
	Error=> , 
	ErrorID=> );
	
axis_BigGate_Right_Reset(
	Axis:= axis_BigGate_Right, 
	Execute:= bAxis_BigGate_Right_Reset, 
	Done=> , 
	Busy=> , 
	Error=> , 
	ErrorID=> );
	

//小龙门
axis_SmallGate_Left_Reset(
	Axis:= axis_SmallGate_Left, 
	Execute:= bAxis_SmallGate_Left_Reset, 
	Done=> , 
	Busy=> , 
	Error=> , 
	ErrorID=> );
	
axis_SmallGate_Right_Reset(
	Axis:= axis_SmallGate_Right, 
	Execute:= bAxis_SmallGate_Right_Reset, 
	Done=> , 
	Busy=> , 
	Error=> , 
	ErrorID=> );

	
	
//后龙门
axis_BackGate_Left_Reset(
	Axis:= axis_BackGate_Left, 
	Execute:= bAxis_BackGate_Left_Reset, 
	Done=> , 
	Busy=> , 
	Error=> , 
	ErrorID=> );
	
axis_BackGate_Right_Reset(
	Axis:= axis_BackGate_Right, 
	Execute:= bAxis_BackGate_Right_Reset, 
	Done=> , 
	Busy=> , 
	Error=> , 
	ErrorID=> );

END_PROGRAM

// ---- POUs/AxisStop.TcPOU
PROGRAM AxisStop
VAR
	i				:USINT := 1;
END_VAR

//IF NOT bEmergencyStopBtn THEN
//	bAxis_All_Stop := TRUE;
//ELSE
//	bAxis_All_Stop := FALSE;
	
//END_IF


// 所有轴停止
//IF bAxis_All_Stop THEN
//	FOR i:=1 TO nAxisNum DO
//		aAxis_All_Stop_Group[i]^ := TRUE;
//	END_FOR
//ELSE
//	FOR i:=1 TO nAxisNum DO
//		aAxis_All_Stop_Group[i]^ := FALSE;
//	END_FOR
//END_IF



// LeftArm_Left_McStop
axis_LeftArm_Left_McStop(
	Axis:= axis_LeftArm_Left, 
	Execute:= bAxis_LeftArm_Left_McStop OR bAxis_All_Stop OR NOT bEmergencyStopBtn, 
	Deceleration:= , 
	Jerk:= , 
	Options:= , 
	Done=> , 
	Busy=> , 
	Active=> , 
	CommandAborted=> , 
	Error=> , 
	ErrorID=> );
	
// LeftArm_Right_McStop
axis_LeftArm_Right_McStop(
	Axis:= axis_LeftArm_Right, 
	Execute:= bAxis_LeftArm_Right_McStop OR bAxis_All_Stop OR NOT bEmergencyStopBtn, 
	Deceleration:= , 
	Jerk:= , 
	Options:= , 
	Done=> , 
	Busy=> , 
	Active=> , 
	CommandAborted=> , 
	Error=> , 
	ErrorID=> );
	
// LeftArm_Wrist_McStop	
axis_LeftArm_Wrist_McStop(
	Axis:= axis_LeftArm_Wrist, 
	Execute:= bAxis_LeftArm_Wrist_McStop OR bAxis_All_Stop OR NOT bEmergencyStopBtn, 
	Deceleration:= , 
	Jerk:= , 
	Options:= , 
	Done=> , 
	Busy=> , 
	Active=> , 
	CommandAborted=> , 
	Error=> , 
	ErrorID=> );

// LeftArm_Lift_McStop		
axis_LeftArm_Lift_McStop(
	Axis:= axis_LeftArm_Lift, 
	Execute:= bAxis_LeftArm_Lift_McStop OR bAxis_All_Stop OR NOT bEmergencyStopBtn, 
	Deceleration:= , 
	Jerk:= , 
	Options:= , 
	Done=> , 
	Busy=> , 
	Active=> , 
	CommandAborted=> , 
	Error=> , 
	ErrorID=> );

	
// RightArm_Left_McStop
axis_RightArm_Left_McStop(
	Axis:= axis_RightArm_Left, 
	Execute:= bAxis_RightArm_Left_McStop OR bAxis_All_Stop OR NOT bEmergencyStopBtn, 
	Deceleration:= , 
	Jerk:= , 
	Options:= , 
	Done=> , 
	Busy=> , 
	Active=> , 
	CommandAborted=> , 
	Error=> , 
	ErrorID=> );
	
// RightArm_Right_McStop
axis_RightArm_Right_McStop(
	Axis:= axis_RightArm_Right, 
	Execute:= bAxis_RightArm_Right_McStop OR bAxis_All_Stop OR NOT bEmergencyStopBtn, 
	Deceleration:= , 
	Jerk:= , 
	Options:= , 
	Done=> , 
	Busy=> , 
	Active=> , 
	CommandAborted=> , 
	Error=> , 
	ErrorID=> );
	
// RightArm_Wrist_McStop	
axis_RightArm_Wrist_McStop(
	Axis:= axis_RightArm_Wrist, 
	Execute:= bAxis_RightArm_Wrist_McStop OR bAxis_All_Stop OR NOT bEmergencyStopBtn, 
	Deceleration:= , 
	Jerk:= , 
	Options:= , 
	Done=> , 
	Busy=> , 
	Active=> , 
	CommandAborted=> , 
	Error=> , 
	ErrorID=> );

// RightArm_Lift_McStop		
axis_RightArm_Lift_McStop(
	Axis:= axis_RightArm_Lift, 
	Execute:= bAxis_RightArm_Lift_McStop OR bAxis_All_Stop OR NOT bEmergencyStopBtn, 
	Deceleration:= , 
	Jerk:= , 
	Options:= , 
	Done=> , 
	Busy=> , 
	Active=> , 
	CommandAborted=> , 
	Error=> , 
	ErrorID=> );

// BigGate_Left_McStop	
axis_BigGate_Left_McStop(
	Axis:= axis_BigGate_Left, 
	Execute:= bAxis_BigGate_Left_McStop OR bAxis_All_Stop OR NOT bEmergencyStopBtn, 
	Deceleration:= , 
	Jerk:= , 
	Options:= , 
	Done=> , 
	Busy=> , 
	Active=> , 
	CommandAborted=> , 
	Error=> , 
	ErrorID=> );
	
// BigGate_Right_McStop
axis_BigGate_Right_McStop(
	Axis:= axis_BigGate_Right, 
	Execute:= bAxis_BigGate_Right_McStop OR bAxis_All_Stop OR NOT bEmergencyStopBtn, 
	Deceleration:= , 
	Jerk:= , 
	Options:= , 
	Done=> , 
	Busy=> , 
	Active=> , 
	CommandAborted=> , 
	Error=> , 
	ErrorID=> );
	
// SmallGate_Left_McStop	
axis_SmallGate_Left_McStop(
	Axis:= axis_SmallGate_Left, 
	Execute:= bAxis_SmallGate_Left_McStop OR bAxis_All_Stop OR NOT bEmergencyStopBtn, 
	Deceleration:= , 
	Jerk:= , 
	Options:= , 
	Done=> , 
	Busy=> , 
	Active=> , 
	CommandAborted=> , 
	Error=> , 
	ErrorID=> );
	
// SmallGate_Right_McStop
axis_SmallGate_Right_McStop(
	Axis:= axis_SmallGate_Right, 
	Execute:= bAxis_SmallGate_Right_McStop OR bAxis_All_Stop OR NOT bEmergencyStopBtn, 
	Deceleration:= , 
	Jerk:= , 
	Options:= , 
	Done=> , 
	Busy=> , 
	Active=> , 
	CommandAborted=> , 
	Error=> , 
	ErrorID=> );
	
	
// BackGate_Left_McStop	
axis_BackGate_Left_McStop(
	Axis:= axis_BackGate_Left, 
	Execute:= bAxis_BackGate_Left_McStop OR bAxis_All_Stop OR NOT bEmergencyStopBtn, 
	Deceleration:= , 
	Jerk:= , 
	Options:= , 
	Done=> , 
	Busy=> , 
	Active=> , 
	CommandAborted=> , 
	Error=> , 
	ErrorID=> );
	
// BackGate_Right_McStop
axis_BackGate_Right_McStop(
	Axis:= axis_BackGate_Right, 
	Execute:= bAxis_BackGate_Right_McStop OR bAxis_All_Stop OR NOT bEmergencyStopBtn, 
	Deceleration:= , 
	Jerk:= , 
	Options:= , 
	Done=> , 
	Busy=> , 
	Active=> , 
	CommandAborted=> , 
	Error=> , 
	ErrorID=> );
	
axis_LeftWheel_Steer_McStop(
	Axis:= axis_LeftWheel_Steer, 
	Execute:= bAxis_LeftWheel_Steer_McStop OR bAxis_All_Stop OR NOT bEmergencyStopBtn, 
	Deceleration:= , 
	Jerk:= , 
	Options:= , 
	Done=> , 
	Busy=> , 
	Active=> , 
	CommandAborted=> , 
	Error=> , 
	ErrorID=> );
	
axis_LeftWheel_Walk_McStop(
	Axis:= axis_LeftWheel_Walk, 
	Execute:= bAxis_LeftWheel_Walk_McStop OR bAxis_All_Stop OR NOT bEmergencyStopBtn, 
	Deceleration:= , 
	Jerk:= , 
	Options:= , 
	Done=> , 
	Busy=> , 
	Active=> , 
	CommandAborted=> , 
	Error=> , 
	ErrorID=> );
	
axis_RightWheel_Steer_McStop(
	Axis:= axis_RightWheel_Steer, 
	Execute:= bAxis_RightWheel_Steer_McStop OR bAxis_All_Stop OR NOT bEmergencyStopBtn, 
	Deceleration:= , 
	Jerk:= , 
	Options:= , 
	Done=> , 
	Busy=> , 
	Active=> , 
	CommandAborted=> , 
	Error=> , 
	ErrorID=> );
	
axis_RightWheel_Walk_McStop(
	Axis:= axis_RightWheel_Walk, 
	Execute:= bAxis_RightWheel_Walk_McStop OR bAxis_All_Stop OR NOT bEmergencyStopBtn, 
	Deceleration:= , 
	Jerk:= , 
	Options:= , 
	Done=> , 
	Busy=> , 
	Active=> , 
	CommandAborted=> , 
	Error=> , 
	ErrorID=> );

END_PROGRAM

// ---- POUs/GateMove.TcPOU
PROGRAM GateMove
VAR
	
	(* 大龙门 *)
	bigGateGearIn			:MC_GearIn;				// 大龙门电子齿轮，LeftAxis为Master
	bigGateGearOut			:MC_GearOut;			// 大龙门电子齿轮取消啮合
	bigGateLeftAxisJog		:MC_Jog;				// 大龙门Jog(实际上电子齿轮的Master轴axis_BigGate_Left的Mc_Jog)
	bigGateLeftAxisMoveAbs	:MC_MoveAbsolute;		// 大龙门MoveAbs(实际上电子齿轮的Master轴axis_BigGate_Left的Mc_MoveAbsolute)
	
	// 当激活大龙门左轴或者右轴的手动控制时bManualCtrl_Part_BigGate_Left或bManualCtrl_Part_BigGate_Right为True，会把此变量置false
	//bBigGate_Gearin_do				:BOOL:=TRUE;			
	
	nBigGate_Speed					:LREAL:=2;		// 大龙门移动速度
	nBigGate_MoveAbs_TarPos			:LREAL;			// 大龙门MoveAbs目标位置
	
	
	
	(* 小龙门 *)
	smallGateGearIn				:MC_GearIn;				// 小龙门电子齿轮，LeftAxis为Master
	smallGateGearOut			:MC_GearOut;			// 小龙门电子齿轮取消啮合
	smallGateLeftAxisJog		:MC_Jog;				// 小龙门左轴(电子齿轮的Master轴)MC_Jog
	smallGateLeftAxisMoveAbs	:MC_MoveAbsolute;		// 小龙门MoveAbs(实际上电子齿轮的Master轴axis_SmallGate_Left的Mc_MoveAbsolute)
	
	// 默认为啮合状态，当激活大龙门左轴或者右轴的手动控制时bManualCtrl_Part_SmallGate_Left为true
	//或bManualCtrl_Part_SmallGate_Right为True，会把此变量置false
	//bSmallGate_Gearin_do		:BOOL:=TRUE;
	
	nSmallGate_Speed					:LREAL:=2;		// 小龙门移动速度
	nSmallGate_MoveAbs_TarPos			:LREAL;			// 小龙门MoveAbs目标位置
	
	
	
	(*后龙门*)
		backGateGearIn					:MC_GearIn;
	backGateGearOut					:MC_GearOut;	                    			
	backGateLeftAxisJog 			:MC_Jog;
	backGateLeftAxisMoveAbs			:MC_MoveAbsolute;		// 后龙门MoveAbs(实际上电子齿轮的Master轴axis_BackGate_Left的Mc_MoveAbsolute)                    			
	
	//bBackGate_Gearin_do				:BOOL:=TRUE;

	nBackGate_Speed					:LREAL:=5;		// 后龙门移动速度
	nBackGate_MoveAbs_TarPos		:LREAL;			// 后龙门MoveAbs目标位置	
	
	
END_VAR



// 当恢复停止按钮或者急停时,大小后龙门需要重新啮合一下电子齿轮
IF bAxis_All_Stop OR NOT bEmergencyStopBtn THEN
	bSmallGate_Gearin_do	:=	FALSE;
    bBigGate_Gearin_do		:=	FALSE;
    bBackGate_Gearin_do		:=	FALSE;
ELSE
	bSmallGate_Gearin_do	:=	TRUE;
    bBigGate_Gearin_do		:=	TRUE;
    bBackGate_Gearin_do		:=	TRUE;
END_IF


IF bManualCtrl_Part_BigGate_Left OR bManualCtrl_Part_BigGate_Right THEN
	bBigGate_Gearin_do		:=	FALSE;
END_IF

IF bManualCtrl_Part_SmallGate_Left OR bManualCtrl_Part_SmallGate_Right THEN
	bSmallGate_Gearin_do		:=	FALSE;
END_IF

IF bManualCtrl_Part_BackGate_Left OR bManualCtrl_Part_BackGate_Right THEN
	bBackGate_Gearin_do		:=	FALSE;
END_IF


// BigGate Mc_Jog
bigGateLeftAxisJog(
	Axis:= axis_BigGate_Left, 
	JogForward:= bBigGate_Up AND bManualCtrl_Asm_BigGate, 
	JogBackwards:= bBigGate_Down AND bManualCtrl_Asm_BigGate, 
	Mode:= MC_JOGMODE_CONTINOUS, 
	Position:= , 
	Velocity:= nBigGate_Speed, 
	Acceleration:= , 
	Deceleration:= , 
	Jerk:= , 
	Done=> , 
	Busy=> , 
	Active=> , 
	CommandAborted=> , 
	Error=> , 
	ErrorID=> );
	
// BigGate Mc_Absolute	
bigGateLeftAxisMoveAbs(
	Axis:= axis_BigGate_Left, 
	Execute:= bBigGate_MoveAbs AND bManualCtrl_Asm_BigGate, 
	Position:= nBigGate_MoveAbs_TarPos, 
	Velocity:= nBigGate_Speed, 
	Acceleration:= , 
	Deceleration:= , 
	Jerk:= , 
	BufferMode:= , 
	Options:= , 
	Done=> , 
	Busy=> , 
	Active=> , 
	CommandAborted=> , 
	Error=> , 
	ErrorID=> );


bigGateGearIn(
	Master:= axis_BigGate_Left, 
	Slave:= axis_BigGate_Right , 
	Execute:= bBigGate_Gearin_do, 
	RatioNumerator:=-1 , 
	RatioDenominator:=1 , 
	Acceleration:= , 
	Deceleration:= , 
	Jerk:= , 
	BufferMode:= , 
	Options:= , 
	InGear=> , 
	Busy=> , 
	Active=> , 
	CommandAborted=> , 
	Error=> , 
	ErrorID=> );
	
	
bigGateGearOut(
	Slave:=axis_BigGate_Right , 
	Execute:= NOT bBigGate_Gearin_do, 
	Options:= , 
	Done=> , 
	Busy=> , 
	Error=> , 
	ErrorID=> );
	
	
	
	
	
	
	
	
// SmallGate Mc_Jog
smallGateLeftAxisJog(
	Axis:= axis_SmallGate_Left, 
	JogForward:= bSmallGate_Down AND bManualCtrl_Asm_SmallGate, 
	JogBackwards:= bSmallGate_Up AND bManualCtrl_Asm_SmallGate, 
	Mode:= MC_JOGMODE_CONTINOUS, 
	Position:= , 
	Velocity:= nSmallGate_Speed, 
	Acceleration:= , 
	Deceleration:= , 
	Jerk:= , 
	Done=> , 
	Busy=> , 
	Active=> , 
	CommandAborted=> , 
	Error=> , 
	ErrorID=> );

// SmallGate Mc_MoveAbsolute
smallGateLeftAxisMoveAbs(
	Axis:= axis_SmallGate_Left, 
	Execute:= bSmallGate_MoveAbs AND bManualCtrl_Asm_SmallGate, 
	Position:= (-1)*nSmallGate_MoveAbs_TarPos, 						// 反转升，所以绝对位置也要反着
	Velocity:= nSmallGate_Speed, 
	Acceleration:= , 
	Deceleration:= , 
	Jerk:= , 
	BufferMode:= , 
	Options:= , 
	Done=> , 
	Busy=> , 
	Active=> , 
	CommandAborted=> , 
	Error=> , 
	ErrorID=> );
	
smallGateGearIn(
	Master:= axis_SmallGate_Left, 
	Slave:= axis_SmallGate_Right, 
	Execute:= bSmallGate_Gearin_do, 
	RatioNumerator:= -1, 
	RatioDenominator:= 1, 
	Acceleration:= , 
	Deceleration:= , 
	Jerk:= , 
	BufferMode:= , 
	Options:= , 
	InGear=> , 
	Busy=> , 
	Active=> , 
	CommandAborted=> , 
	Error=> , 
	ErrorID=> );
	
	
smallGateGearOut(
	Slave:= axis_SmallGate_Right, 
	Execute:= NOT bSmallGate_Gearin_do, 
	Options:= , 
	Done=> , 
	Busy=> , 
	Error=> , 
	ErrorID=> );	

	
	
	
	
	
	
// Mc_Jog
backGateLeftAxisJog(
	Axis:= axis_BackGate_Left, 
	JogForward:= bBackGate_Down AND bManualCtrl_Asm_BackGate, 
	JogBackwards:= bBackGate_Up AND bManualCtrl_Asm_BackGate, 
	Mode:= MC_JOGMODE_CONTINOUS, 
	Position:= , 
	Velocity:= nBackGate_Speed, 
	Acceleration:= , 
	Deceleration:= , 
	Jerk:= , 
	Done=> , 
	Busy=> , 
	Active=> , 
	CommandAborted=> , 
	Error=> , 
	ErrorID=> );

// Mc_MoveAbs
backGateLeftAxisMoveAbs(
	Axis:= axis_BackGate_Left, 
	Execute:= bBackGate_MoveAbs AND bManualCtrl_Asm_BackGate, 
	Position:= (-1)*nBackGate_MoveAbs_TarPos, 						// 反转升，所以绝对位置也要反着
	Velocity:= nBackGate_Speed, 
	Acceleration:= , 
	Deceleration:= , 
	Jerk:= , 
	BufferMode:= , 
	Options:= , 
	Done=> , 
	Busy=> , 
	Active=> , 
	CommandAborted=> , 
	Error=> , 
	ErrorID=> );	

	
backGateGearIn(
	Master:= axis_BackGate_Left, 
	Slave:= axis_BackGate_Right, 
	Execute:= bBackGate_GearIn_do, 
	RatioNumerator:= 1, 
	RatioDenominator:= 1, 
	Acceleration:= , 
	Deceleration:= , 
	Jerk:= , 
	BufferMode:= , 
	Options:= , 
	InGear=> , 
	Busy=> , 
	Active=> , 
	CommandAborted=> , 
	Error=> , 
	ErrorID=> );


backGateGearOut(
	Slave:= axis_BackGate_Right, 
	Execute:= NOT bBackGate_GearIn_do, 
	Options:= , 
	Done=> , 
	Busy=> , 
	Error=> , 
	ErrorID=> );

END_PROGRAM

// ---- POUs/LeftArmManualCtrlMove.TcPOU
PROGRAM LeftArmManualCtrlMove
VAR
	
	point												:Points;					// 当前腕关节坐标
	target_angle										:Angles;					// 臂左右电机目标角度
	manualState											:USINT;						// 手动控制状态标志位，0
	speed												:REAL := 0.5;					// 笛卡尔坐标位移速度
	x													:REAL;						// 腕关节目标位置x
	y													:REAL;						// 腕关节目标位置y
	wrist_angle											:REAL;						// 腕电机角度
	
	//左臂举升电机
	LeftArm_Lift_Jog									:MC_Jog;
	bLeftArm_Lift_Up									:BOOL;
	bLeftArm_Lift_Down									:BOOL;
	nLeftArmLiftSpeed									:LREAL:=3;					//举升电机速度
	
	LeftArm_Right_ExtPosGen_Enable						:MC_ExtSetPointGenEnable;
	LeftArm_Right_ExtPosGen_Disable                     :MC_ExtSetPointGenDisable;
	LeftArm_Left_ExtPosGen_Enable                       :MC_ExtSetPointGenEnable;
	LeftArm_Left_ExtPosGen_Disable	                    :MC_ExtSetPointGenDisable;
	LeftArm_Wrist_ExtPosGen_Enable                      :MC_ExtSetPointGenEnable;
	LeftArm_Wrist_ExtPosGen_Disable	                    :MC_ExtSetPointGenDisable;
	
	//串口
	//fb_SerialCom		:FB_SerialCom;					
	//wrist_angle_int		:INT;
	//wrist_angle_byte	:BYTE;
	
	
END_VAR

axis_LeftArm_Left();
axis_LeftArm_Right();
axis_LeftArm_Wrist();
ExtPosGen();


// 外部位置发生器失能
LeftArm_Right_ExtPosGen_Enable.Execute 		:= FALSE;
LeftArm_Right_ExtPosGen_Disable.Execute 	:= FALSE;
LeftArm_Left_ExtPosGen_Enable.Execute 		:= FALSE;
LeftArm_Left_ExtPosGen_Disable.Execute 		:= FALSE;
LeftArm_Wrist_ExtPosGen_Enable.Execute 		:= FALSE;
LeftArm_Wrist_ExtPosGen_Disable.Execute 	:= FALSE;

IF bManualCtrl_Asm_LeftArm THEN
	// 举升电机McJog
	LeftArmLiftJog();
	
	// 运动学正解出当前腕关节点坐标
	point := LeftArmFK(axis_LeftArm_Right.NcToPlc.ActPos, axis_LeftArm_Left.NcToPlc.ActPos);
	
	// 用舵机进行程序验证的串口背景通讯
	//BackgroundSerialCtrl();
	
	IF bAutoCtrl_Part_LeftWrist THEN
		
		wrist_angle := LeftArmWristIK(axis_LeftArm_Right.NcToPlc.ActPos, axis_LeftArm_Left.NcToPlc.ActPos);		// 逆解出腕电机角度

	END_IF
	

	IF bLeftArm_Forward THEN
		x := point.x;
		y := point.y + speed;
		target_angle := LeftArmIK(x, y);
		manualState := 1;
		
	ELSIF bLeftArm_Backward THEN
	
		x := point.x;
		y := point.y - speed;
		target_angle := LeftArmIK(x, y);
		manualState := 1;
		
	ELSIF bLeftArm_Left THEN
		
		x := point.x - speed;
		y := point.y;
		target_angle := LeftArmIK(x, y);
		manualState := 1;
		
	ELSIF bLeftArm_Right THEN
		
		x := point.x + speed;
		y := point.y;
		target_angle := LeftArmIK(x, y);
		manualState := 1;
		
	ELSE
		manualState := 0;
	END_IF
	
	
	
	CASE manualState OF
		0:
			LeftArm_Right_ExtPosGen_Enable.Execute 		:= FALSE;
			LeftArm_Right_ExtPosGen_Disable.Execute 	:= TRUE;
			LeftArm_Left_ExtPosGen_Enable.Execute 		:= FALSE;
			LeftArm_Left_ExtPosGen_Disable.Execute 		:= TRUE;
			LeftArm_Wrist_ExtPosGen_Enable.Execute 		:= FALSE;
			LeftArm_Wrist_ExtPosGen_Disable.Execute 	:= TRUE;
		
		1:
			LeftArm_Right_ExtPosGen_Enable.Execute := TRUE;
			LeftArm_Left_ExtPosGen_Enable.Execute := TRUE;
			LeftArm_Wrist_ExtPosGen_Enable.Execute := TRUE;
			IF axis_LeftArm_Right.Status.ExtSetPointGenEnabled AND axis_LeftArm_Left.Status.ExtSetPointGenEnabled AND axis_LeftArm_Wrist.Status.ExtSetPointGenEnabled THEN
				MC_ExtSetPointGenFeed(
					Position:= target_angle.theta1_right, 
					Velocity:= 1,  
					Acceleration:= 3,  
					Direction:= 1, 
					Axis:= axis_LeftArm_Right);
		
				MC_ExtSetPointGenFeed(
					Position:= target_angle.theta2_left, 
					Velocity:= 1,  
					Acceleration:= 3,  
					Direction:= 1, 
					Axis:= axis_LeftArm_Left);
					
				MC_ExtSetPointGenFeed(
					Position:= wrist_angle, 
					Velocity:= 1, 
					Acceleration:= 3, 
					Direction:= 1, 
					Axis:= axis_LeftArm_Wrist);
			END_IF
	END_CASE

//ELSE

END_IF

ACTION ExtPosGen:
LeftArm_Right_ExtPosGen_Enable(
	Axis:= axis_LeftArm_Right, 
	Execute:= LeftArm_Right_ExtPosGen_Enable.Execute, 
	Position:= , 
	PositionType:= , 
	Done=> , 
	Busy=> , 
	Error=> , 
	ErrorID=> , 
	Enabled=> );
	
LeftArm_Right_ExtPosGen_Disable(
	Axis:= axis_LeftArm_Right, 
	Execute:= LeftArm_Right_ExtPosGen_Disable.Execute, 
	Done=> , 
	Busy=> , 
	Error=> , 
	ErrorID=> , 
	Enabled=> );
	
LeftArm_Left_ExtPosGen_Enable(
	Axis:= axis_LeftArm_Left, 
	Execute:= LeftArm_Left_ExtPosGen_Enable.Execute, 
	Position:= , 
	PositionType:= , 
	Done=> , 
	Busy=> , 
	Error=> , 
	ErrorID=> , 
	Enabled=> );
	
LeftArm_Left_ExtPosGen_Disable(
	Axis:= axis_LeftArm_Left, 
	Execute:= LeftArm_Left_ExtPosGen_Disable.Execute, 
	Done=> , 
	Busy=> , 
	Error=> , 
	ErrorID=> , 
	Enabled=> );
	
LeftArm_Wrist_ExtPosGen_Enable(
	Axis:= axis_LeftArm_Wrist, 
	Execute:= LeftArm_Wrist_ExtPosGen_Enable.Execute, 
	Position:= , 
	PositionType:= , 
	Done=> , 
	Busy=> , 
	Error=> , 
	ErrorID=> , 
	Enabled=> );
	
LeftArm_Wrist_ExtPosGen_Disable(
	Axis:= axis_LeftArm_Wrist, 
	Execute:= LeftArm_Wrist_ExtPosGen_Disable.Execute, 
	Done=> , 
	Busy=> , 
	Error=> , 
	ErrorID=> , 
	Enabled=> );
END_ACTION

ACTION LeftArmLiftJog:
LeftArm_Lift_Jog(
	Axis:= axis_LeftArm_Lift, 
	JogForward:= bLeftArm_Lift_Up, 
	JogBackwards:= bLeftArm_Lift_Down, 
	Mode:= MC_JOGMODE_CONTINOUS, 
	Position:= , 
	Velocity:= nLeftArmLiftSpeed, 
	Acceleration:= , 
	Deceleration:= , 
	Jerk:= , 
	Done=> , 
	Busy=> , 
	Active=> , 
	CommandAborted=> , 
	Error=> , 
	ErrorID=> );
END_ACTION

END_PROGRAM

// ---- POUs/LeftArmFK.TcPOU
FUNCTION LeftArmFK : Points
VAR_INPUT
	theta1:LREAL;
	theta2:LREAL;
END_VAR
VAR
	// 中间变量
	theta1_rad:LREAL;
	theta2_rad:LREAL;
	rr:LREAL;						//r变量被倍福占用了，所以此处用rr
	u:LREAL;
	angle_ACD:LREAL;
	angle_DCE:LREAL;
	angle_ACF:LREAL;
	angle_FCG:LREAL;
	angle_FCI:LREAL;
	
	// 输出
	points : Points;

END_VAR

theta1_rad := DEG_TO_RAD(theta1);
theta2_rad := DEG_TO_RAD(theta2);


rr := SQRT(EXPT((2*LeftArm_w+LeftArm_f*COS(theta1_rad)-LeftArm_g*COS(theta2_rad)),2) + EXPT((LeftArm_f*SIN(theta1_rad)-LeftArm_g*SIN(theta2_rad)),2));  

u := SQRT(EXPT((2*LeftArm_w-LeftArm_g*COS(theta2_rad)),2) + EXPT((-LeftArm_g*SIN(theta2_rad)),2));


angle_ACD := ACOS((rr*rr+LeftArm_f*LeftArm_f-u*u)/(2*rr*LeftArm_f));


angle_DCE := ACOS((rr*rr + LeftArm_i*LeftArm_i -LeftArm_h*LeftArm_h)/(2*rr*LeftArm_i));


angle_ACF := angle_ACD + angle_DCE + DEG_TO_RAD(LeftArm_angle_FCE);


angle_FCG := angle_ACF - theta1_rad;


angle_FCI := PI - angle_FCG;
points.x := LeftArm_w + LeftArm_f*COS(theta1_rad) + LeftArm_n*COS(angle_FCI);
points.y := LeftArm_f*SIN(theta1_rad) + LeftArm_n*SIN(angle_FCI);

LeftArmFK := points;

END_FUNCTION

// ---- POUs/LeftArmWristIK.TcPOU
FUNCTION LeftArmWristIK : REAL
VAR_INPUT
	theta1:LREAL;					// 左臂右电机角度
	theta2:LREAL;					// 左臂左电机角度
END_VAR
VAR
	// 中间变量
	theta1_rad:LREAL;
	theta2_rad:LREAL;
	rr:LREAL;						//r变量被倍福占用了，所以此处用rr
	u:LREAL;
	angle_ACD:LREAL;
	angle_DCE:LREAL;
	angle_ACE:LREAL;
	angle_ECG:LREAL;
	angle_ECI:LREAL;
	
	point_E:Points;
	point_F:Points;
	
	jx:REAL;				//EF向量的横坐标
	jy:REAL;				//EF向量的纵坐标
	vx:REAL:=0;				//+y单位向量的横坐标
	vy:REAL:=1;				//+y单位向量的纵坐标
	result_cross:REAL;		//EF向量和+y向量的叉乘结果
	
	angle_Beta:REAL;
	
	
END_VAR

theta1_rad := DEG_TO_RAD(theta1);
theta2_rad := DEG_TO_RAD(theta2);

point_F := LeftArmFK(theta1, theta2);

rr := SQRT(EXPT((2*LeftArm_w+LeftArm_f*COS(theta1_rad)-LeftArm_g*COS(theta2_rad)),2) + EXPT((LeftArm_f*SIN(theta1_rad)-LeftArm_g*SIN(theta2_rad)),2));  

u := SQRT(EXPT((2*LeftArm_w-LeftArm_g*COS(theta2_rad)),2) + EXPT((-LeftArm_g*SIN(theta2_rad)),2));

angle_ACD := ACOS((rr*rr+LeftArm_f*LeftArm_f-u*u)/(2*rr*LeftArm_f));

angle_DCE := ACOS((rr*rr + LeftArm_i*LeftArm_i -LeftArm_h*LeftArm_h)/(2*rr*LeftArm_i));

angle_ACE := angle_ACD + angle_DCE;

angle_ECG := angle_ACE - theta1_rad;
    
angle_ECI := PI - angle_ECG;

point_E.x := LeftArm_w + LeftArm_f*COS(theta1_rad) + LeftArm_i*COS(angle_ECI);
point_E.y := LeftArm_f*SIN(theta1_rad) + LeftArm_i*SIN(angle_ECI);

jx := point_F.x - point_E.x;
jy := point_F.y - point_E.y;

result_cross := jx*vy - jy*vx;

IF result_cross > 0 THEN
	angle_Beta := ACOS((jx*vx+jy*vy)/(SQRT(jx*jx+jy*jy)*SQRT(vx*vx+vy*vy)));
ELSIF result_cross < 0 THEN
	angle_Beta := -ACOS((jx*vx+jy*vy)/(SQRT(jx*jx+jy*jy)*SQRT(vx*vx+vy*vy)));
ELSE
	angle_Beta := 0;
END_IF

LeftArmWristIK := RAD_TO_DEG(angle_Beta);

END_FUNCTION

// ---- POUs/LeftArmIK.TcPOU
FUNCTION LeftArmIK : Angles
VAR_INPUT
	x:LREAL;
	y:LREAL;
END_VAR
VAR
	
	// 中间量
	p:LREAL;
	q:LREAL;
	l:LREAL;
	k:LREAL;
	angle_CAF:LREAL;	
	angle_OAF:LREAL;
	theta1:LREAL;
	theta2:LREAL;
	angle_ACF:LREAL;
	angle_ACE:LREAL;
	angle_CAE:LREAL;
	angle_EAB:LREAL;
	angle_EBA:LREAL;
	angle_DBE:LREAL;
	
	// 输出
	angles		:Angles;
	
END_VAR

// TWINCAT 角度换算以弧度为单位

p := SQRT((x-LeftArm_w)*(x-LeftArm_w)+y*y);
q := SQRT(x*x + y*y);
 
//n := SQRT(i*i+j*j-2*i*j*COS(DEG_TO_RAD(angle_a)));
angle_CAF := ACOS((LeftArm_f*LeftArm_f+p*p-LeftArm_n*LeftArm_n)/(2*LeftArm_f*p));
angle_OAF := ACOS((LeftArm_w*LeftArm_w+p*p-q*q)/(2*LeftArm_w*p));
theta1 := PI-angle_CAF-angle_OAF;

angle_ACF := ACOS((LeftArm_f*LeftArm_f+LeftArm_n*LeftArm_n-p*p)/(2*LeftArm_f*LeftArm_n));
//angle_FCE := ACOS((n*n+i*i-j*j)/(2*n*i));
angle_ACE := angle_ACF - DEG_TO_RAD(LeftArm_angle_FCE);
l := SQRT(LeftArm_i*LeftArm_i+LeftArm_f*LeftArm_f-2*LeftArm_i*LeftArm_f*COS(angle_ACE));
angle_CAE := ACOS((LeftArm_f*LeftArm_f+l*l-LeftArm_i*LeftArm_i)/(2*LeftArm_f*l));
angle_EAB := PI-theta1 - angle_CAE;
k := SQRT(l*l + 4*LeftArm_w*LeftArm_w - 4*l*LeftArm_w*COS(angle_EAB));
angle_EBA := ACOS((k*k+4*LeftArm_w*LeftArm_w-l*l)/(4*k*LeftArm_w));
angle_DBE := ACOS((LeftArm_g*LeftArm_g+k*k-LeftArm_h*LeftArm_h)/(2*LeftArm_g*k));
theta2 := angle_EBA + angle_DBE;

angles.theta1_right := RAD_TO_DEG(theta1);
angles.theta2_left := RAD_TO_DEG(theta2);


LeftArmIK := angles;

END_FUNCTION

// ---- POUs/MAIN.TcPOU
PROGRAM MAIN
VAR
	
	a1			:INT		:=100;
	b2			:BOOL		:=FALSE;
	c3 			:LREAL 		:= 0;
	
	er			:DWORD;
	er1         :DWORD;
	
	arrLeftBoxStack	:ARRAY[1..50] OF BOX;
	arrRightBoxStack:ARRAY[1..50] OF BOX;
	
	
	//er:=axis_SmallGate_Left.NcToPlc.StateDWord

END_VAR

axis_BigGate_Left();	
er := axis_BigGate_Left.NcToPlc.StateDWord AND SHL(16#1, 28);
er1:= axis_BigGate_Left.NcToPlc.StateDWord AND SHL(16#1, 31);

END_PROGRAM

// ---- POUs/MoveExtPos.TcPOU
PROGRAM MoveExtPos
VAR
	armState	:UINT:=0;
	chabustate	:UINT:=0;
	
	LeftArm_Right_ExtPosGen_Enable						:MC_ExtSetPointGenEnable;
	LeftArm_Right_ExtPosGen_Disable                     :MC_ExtSetPointGenDisable;
	LeftArm_Left_ExtPosGen_Enable                       :MC_ExtSetPointGenEnable;
	LeftArm_Left_ExtPosGen_Disable	                    :MC_ExtSetPointGenDisable;
	LeftArm_Wrist_ExtPosGen_Enable                      :MC_ExtSetPointGenEnable;
	LeftArm_Wrist_ExtPosGen_Disable	                    :MC_ExtSetPointGenDisable;
	
	RightArm_Right_ExtPosGen_Enable						:MC_ExtSetPointGenEnable;
	RightArm_Right_ExtPosGen_Disable                     :MC_ExtSetPointGenDisable;
	RightArm_Left_ExtPosGen_Enable                       :MC_ExtSetPointGenEnable;
	RightArm_Left_ExtPosGen_Disable	                    :MC_ExtSetPointGenDisable;
	RightArm_Wrist_ExtPosGen_Enable                      :MC_ExtSetPointGenEnable;
	RightArm_Wrist_ExtPosGen_Disable	                    :MC_ExtSetPointGenDisable;
	
	currentPosition_LeftArm				:Points;
	currentPosition_RightArm				:Points;

	//leftpoints						:ARRAY[0..5,0..1] OF LREAL:=[[-80,390],[390,880],[-80,390],[-80,880],[-80,390],[-400,830]];
	//rightpoints						:ARRAY[0..5,0..1] OF LREAL:=[[-80,390],[390,880],[-80,390],[-80,880],[-80,390],[-400,830]];	
	LeftArmWristTargetPos				:REAL;
	RightArmWristTargetPos				:REAL;	
	
	t			:LREAL:=0;
	delta_t		:LREAL:=0.0005;
	
	lx:LREAL;
	ly:LREAL;
	rx:LREAL;
	ry:LREAL;
	
	LeftArmAngle			:Angles;
	RightArmAngle			:Angles;


	
	

END_VAR

axis_LeftArm_Left();
axis_LeftArm_Right();
axis_LeftArm_Wrist();
axis_RightArm_Left();
axis_RightArm_Right();
axis_RightArm_Wrist();
ACT_ExtGen();


// 外部位置发生器失能
LeftArm_Right_ExtPosGen_Enable.Execute 		:= FALSE;
LeftArm_Right_ExtPosGen_Disable.Execute 	:= FALSE;
LeftArm_Left_ExtPosGen_Enable.Execute 		:= FALSE;
LeftArm_Left_ExtPosGen_Disable.Execute 		:= FALSE;
LeftArm_Wrist_ExtPosGen_Enable.Execute 		:= FALSE;
LeftArm_Wrist_ExtPosGen_Disable.Execute 	:= FALSE;	

RightArm_Right_ExtPosGen_Enable.Execute 	:= FALSE;
RightArm_Right_ExtPosGen_Disable.Execute 	:= FALSE;
RightArm_Left_ExtPosGen_Enable.Execute 		:= FALSE;
RightArm_Left_ExtPosGen_Disable.Execute 	:= FALSE;
RightArm_Wrist_ExtPosGen_Enable.Execute 	:= FALSE;
RightArm_Wrist_ExtPosGen_Disable.Execute 	:= FALSE;	


IF bAutoMovePosSet THEN

	
	CASE armState OF
		
		0:// 运动学正解出当前腕关节点坐标
			currentPosition_LeftArm 	:= LeftArmFK(axis_LeftArm_Right.NcToPlc.ActPos, axis_LeftArm_Left.NcToPlc.ActPos);
			currentPosition_RightArm 	:= RightArmFK(axis_RightArm_Right.NcToPlc.ActPos, axis_RightArm_Left.NcToPlc.ActPos);
			LeftArmWristTargetPos		:= LeftArmWristIK(axis_LeftArm_Right.NcToPlc.ActPos, axis_LeftArm_Left.NcToPlc.ActPos);
			RightArmWristTargetPos		:= RightArmWristIK(axis_RightArm_Right.NcToPlc.ActPos, axis_RightArm_Left.NcToPlc.ActPos);
			armState:=1;
		1:// 转动腕关节，到正确的解算位置
			axis_LeftArm_Wrist_MoveAbs(
				Axis:= axis_LeftArm_Wrist, 
				Execute:= TRUE, 
				Position:= LeftArmWristTargetPos, 
				Velocity:= 0.5, 
				Acceleration:= 1, 
				Deceleration:= , 
				Jerk:= , 
				BufferMode:= , 
				Options:= , 
				Done=> , 
				Busy=> , 
				Active=> , 
				CommandAborted=> , 
				Error=> , 
				ErrorID=> );
			
			axis_RightArm_Wrist_MoveAbs(
				Axis:= axis_RightArm_Wrist, 
				Execute:= TRUE, 
				Position:= RightArmWristTargetPos, 
				Velocity:= 0.5, 
				Acceleration:= 1, 
				Deceleration:= , 
				Jerk:= , 
				BufferMode:= , 
				Options:= , 
				Done=> , 
				Busy=> , 
				Active=> , 
				CommandAborted=> , 
				Error=> , 
				ErrorID=> );
			IF axis_RightArm_Wrist_MoveAbs.Done = TRUE AND axis_LeftArm_Wrist_MoveAbs.Done = TRUE THEN
				armState:=2;
			END_IF

			
		2:
			LeftArm_Right_ExtPosGen_Enable.Execute 		:= TRUE;
			LeftArm_Left_ExtPosGen_Enable.Execute 		:= TRUE;
			LeftArm_Wrist_ExtPosGen_Enable.Execute 		:= TRUE;
			RightArm_Right_ExtPosGen_Enable.Execute 	:= TRUE;
			RightArm_Left_ExtPosGen_Enable.Execute 		:= TRUE;
			RightArm_Wrist_ExtPosGen_Enable.Execute 	:= TRUE;
			
			IF axis_LeftArm_Right.Status.ExtSetPointGenEnabled AND axis_LeftArm_Left.Status.ExtSetPointGenEnabled AND axis_RightArm_Right.Status.ExtSetPointGenEnabled AND axis_RightArm_Left.Status.ExtSetPointGenEnabled AND axis_LeftArm_Wrist.Status.ExtSetPointGenEnabled  AND axis_RightArm_Wrist.Status.ExtSetPointGenEnabled THEN

				CASE  chabustate OF
					0:
						lx	:=currentPosition_LeftArm.x+t*(-80-currentPosition_LeftArm.x);
						ly 	:=currentPosition_LeftArm.y+t*(390-currentPosition_LeftArm.y);
						rx	:=currentPosition_RightArm.x+t*(120-currentPosition_RightArm.x);
						ry 	:=currentPosition_RightArm.y+t*(370-currentPosition_RightArm.y);
						t	:= t+delta_t;
						IF t>=1 THEN
							LeftArm_Right_ExtPosGen_Enable.Execute := FALSE;
							LeftArm_Left_ExtPosGen_Enable.Execute := FALSE;
							RightArm_Right_ExtPosGen_Enable.Execute := FALSE;
							RightArm_Left_ExtPosGen_Enable.Execute := FALSE;
							chabustate:=1;
							t	:=0;
						END_IF

					1:

						lx	:=t*470-80;
						ly	:=390+t*490;
						rx	:=120+250*t;
						ry	:=370+510*t;
						t	:= t+delta_t;
						IF t >=1 THEN
							LeftArm_Right_ExtPosGen_Enable.Execute := FALSE;
							LeftArm_Left_ExtPosGen_Enable.Execute := FALSE;
							RightArm_Right_ExtPosGen_Enable.Execute := FALSE;
							RightArm_Left_ExtPosGen_Enable.Execute := FALSE;
							chabustate := 2;
							t:=0;
						END_IF
					2:
						lx	:=390-t*470;
						ly	:=880-t*490;
						rx	:=370-250*t;
						ry	:=880-510*t;
						t	:= t+delta_t;
						IF t>=1 THEN
							LeftArm_Right_ExtPosGen_Enable.Execute := FALSE;
							LeftArm_Left_ExtPosGen_Enable.Execute := FALSE;
							RightArm_Right_ExtPosGen_Enable.Execute := FALSE;
							RightArm_Left_ExtPosGen_Enable.Execute := FALSE;
							chabustate := 3;
							t:=0;
						END_IF
					3:
						lx := -80;
						ly := 390+490*t;
						rx := 120;
						ry := 370+510*t;
						t:=t+delta_t;
						IF t>= 1 THEN
							LeftArm_Right_ExtPosGen_Enable.Execute := FALSE;
							LeftArm_Left_ExtPosGen_Enable.Execute := FALSE;
							RightArm_Right_ExtPosGen_Enable.Execute := FALSE;
							RightArm_Left_ExtPosGen_Enable.Execute := FALSE;
							chabustate	:=4;
							t:=0;
						END_IF
					4:
						lx := -80;
						ly := 880-490*t;
						rx := 120;
						ry := 880-510*t;
						t:= t+delta_t;
						IF t>=1 THEN
							LeftArm_Right_ExtPosGen_Enable.Execute := FALSE;
							LeftArm_Left_ExtPosGen_Enable.Execute := FALSE;
							RightArm_Right_ExtPosGen_Enable.Execute := FALSE;
							RightArm_Left_ExtPosGen_Enable.Execute := FALSE;
							chabustate := 5;
							t:=0;
						END_IF
					5:
						lx := -80-320*t;
						ly := 390+440*t;
						rx := 120-450*t;
						ry := 370+480*t;
						t:=t+delta_t;
						IF t>= 1 THEN
							LeftArm_Right_ExtPosGen_Enable.Execute := FALSE;
							LeftArm_Left_ExtPosGen_Enable.Execute := FALSE;
							RightArm_Right_ExtPosGen_Enable.Execute := FALSE;
							RightArm_Left_ExtPosGen_Enable.Execute := FALSE;
							chabustate	:=6;
							t:=0;
						END_IF
					6:
						lx := -400+320*t;
						ly := 830-440*t;
						rx := -330+450*t;
						ry := 850-480*t;
						t:= t+delta_t;
						IF t>=1 THEN
							LeftArm_Right_ExtPosGen_Enable.Execute := FALSE;
							LeftArm_Left_ExtPosGen_Enable.Execute := FALSE;
							RightArm_Right_ExtPosGen_Enable.Execute := FALSE;
							RightArm_Left_ExtPosGen_Enable.Execute := FALSE;
							chabustate := 1;
							t:=0;
						END_IF

				END_CASE
				
				LeftArmAngle := LeftArmIK(lx,ly);
				LeftArmWristTargetPos := LeftArmWristIK(LeftArmAngle.theta1_right, LeftArmAngle.theta2_left);
				
				RightArmAngle := RightArmIK(rx,ry);
				RightArmWristTargetPos := RightArmWristIK(RightArmAngle.theta1_right, RightArmAngle.theta2_left);
					
	
				
				LeftArm_Right_ExtPosGen_Enable.Execute := TRUE;
				LeftArm_Left_ExtPosGen_Enable.Execute := TRUE;
				RightArm_Right_ExtPosGen_Enable.Execute := TRUE;
				RightArm_Left_ExtPosGen_Enable.Execute := TRUE;
				
				MC_ExtSetPointGenFeed(
					Position:= LeftArmAngle.theta1_right, 
					Velocity:= 0.005,  
					Acceleration:= 0.01,  
					Direction:= 1, 
					Axis:= axis_LeftArm_Right);
		
				MC_ExtSetPointGenFeed(
					Position:= LeftArmAngle.theta2_left, 
					Velocity:= 0.005,  
					Acceleration:= 0.001,  
					Direction:= 1, 
					Axis:= axis_LeftArm_Left);
				
				MC_ExtSetPointGenFeed(
					Position:= RightArmAngle.theta1_right, 
					Velocity:= 0.005,  
					Acceleration:= 0.01,  
					Direction:= 1, 
					Axis:= axis_RightArm_Right);
		
				MC_ExtSetPointGenFeed(
					Position:= RightArmAngle.theta2_left, 
					Velocity:= 0.005,  
					Acceleration:= 0.001,  
					Direction:= 1, 
					Axis:= axis_RightArm_left);
												
				MC_ExtSetPointGenFeed(
					Position:= LeftArmWristTargetPos, 
					Velocity:= 0.5, 
					Acceleration:= 1, 
					Direction:= 1, 
					Axis:= axis_LeftArm_Wrist);

					
				MC_ExtSetPointGenFeed(
					Position:= RightArmWristTargetPos, 
					Velocity:= 5, 
					Acceleration:= 10, 
					Direction:= 1, 
					Axis:= axis_RightArm_Wrist);
				

			END_IF
	
	END_CASE




END_IF

ACTION ACT_ExtGen:
LeftArm_Right_ExtPosGen_Enable(
	Axis:= axis_LeftArm_Right, 
	Execute:= LeftArm_Right_ExtPosGen_Enable.Execute, 
	Position:= , 
	PositionType:= , 
	Done=> , 
	Busy=> , 
	Error=> , 
	ErrorID=> , 
	Enabled=> );
	
LeftArm_Right_ExtPosGen_Disable(
	Axis:= axis_LeftArm_Right, 
	Execute:= LeftArm_Right_ExtPosGen_Disable.Execute, 
	Done=> , 
	Busy=> , 
	Error=> , 
	ErrorID=> , 
	Enabled=> );
	
LeftArm_Left_ExtPosGen_Enable(
	Axis:= axis_LeftArm_Left, 
	Execute:= LeftArm_Left_ExtPosGen_Enable.Execute, 
	Position:= , 
	PositionType:= , 
	Done=> , 
	Busy=> , 
	Error=> , 
	ErrorID=> , 
	Enabled=> );
	
LeftArm_Left_ExtPosGen_Disable(
	Axis:= axis_LeftArm_Left, 
	Execute:= LeftArm_Left_ExtPosGen_Disable.Execute, 
	Done=> , 
	Busy=> , 
	Error=> , 
	ErrorID=> , 
	Enabled=> );
	
LeftArm_Wrist_ExtPosGen_Enable(
	Axis:= axis_LeftArm_Wrist, 
	Execute:= LeftArm_Wrist_ExtPosGen_Enable.Execute, 
	Position:= , 
	PositionType:= , 
	Done=> , 
	Busy=> , 
	Error=> , 
	ErrorID=> , 
	Enabled=> );
	
LeftArm_Wrist_ExtPosGen_Disable(
	Axis:= axis_LeftArm_Wrist, 
	Execute:= LeftArm_Wrist_ExtPosGen_Disable.Execute, 
	Done=> , 
	Busy=> , 
	Error=> , 
	ErrorID=> , 
	Enabled=> );
	
RightArm_Right_ExtPosGen_Enable(
	Axis:= axis_RightArm_Right, 
	Execute:= RightArm_Right_ExtPosGen_Enable.Execute, 
	Position:= , 
	PositionType:= , 
	Done=> , 
	Busy=> , 
	Error=> , 
	ErrorID=> , 
	Enabled=> );
	
RightArm_Right_ExtPosGen_Disable(
	Axis:= axis_RightArm_Right, 
	Execute:= RightArm_Right_ExtPosGen_Disable.Execute, 
	Done=> , 
	Busy=> , 
	Error=> , 
	ErrorID=> , 
	Enabled=> );
	
RightArm_Left_ExtPosGen_Enable(
	Axis:= axis_RightArm_Left, 
	Execute:= RightArm_Left_ExtPosGen_Enable.Execute, 
	Position:= , 
	PositionType:= , 
	Done=> , 
	Busy=> , 
	Error=> , 
	ErrorID=> , 
	Enabled=> );
	
RightArm_Left_ExtPosGen_Disable(
	Axis:= axis_RightArm_Left, 
	Execute:= RightArm_Left_ExtPosGen_Disable.Execute, 
	Done=> , 
	Busy=> , 
	Error=> , 
	ErrorID=> , 
	Enabled=> );
	
RightArm_Wrist_ExtPosGen_Enable(
	Axis:= axis_RightArm_Wrist, 
	Execute:= RightArm_Wrist_ExtPosGen_Enable.Execute, 
	Position:= , 
	PositionType:= , 
	Done=> , 
	Busy=> , 
	Error=> , 
	ErrorID=> , 
	Enabled=> );
	
RightArm_Wrist_ExtPosGen_Disable(
	Axis:= axis_RightArm_Wrist, 
	Execute:= RightArm_Wrist_ExtPosGen_Disable.Execute, 
	Done=> , 
	Busy=> , 
	Error=> , 
	ErrorID=> , 
	Enabled=> );
END_ACTION

END_PROGRAM

// ---- POUs/RightArmFK.TcPOU
FUNCTION RightArmFK : Points
VAR_INPUT
	theta1:LREAL;
	theta2:LREAL;
END_VAR
VAR
	// 中间变量
	theta1_rad:LREAL;
	theta2_rad:LREAL;
	rr:LREAL;						//r变量被倍福占用了，所以此处用rr
	u:LREAL;
	angle_BDC:LREAL;
	angle_CDE:LREAL;
	angle_BDF:LREAL;
	angle_FDG:LREAL;
	
	
	// 输出
	points : Points;

END_VAR

theta1_rad := DEG_TO_RAD(theta1);
theta2_rad := DEG_TO_RAD(theta2);


rr := SQRT(EXPT((2*RightArm_w+RightArm_f*COS(theta1_rad)-RightArm_g*COS(theta2_rad)),2) + EXPT((RightArm_f*SIN(theta1_rad)-RightArm_g*SIN(theta2_rad)),2));  

u := SQRT(EXPT((2*RightArm_w+RightArm_f*COS(theta1_rad)),2) + EXPT((RightArm_f*SIN(theta1_rad)),2));


angle_BDC := ACOS((rr*rr+RightArm_g*RightArm_g-u*u)/(2*rr*RightArm_g));


angle_CDE := ACOS((rr*rr + RightArm_h*RightArm_h -RightArm_i*RightArm_i)/(2*rr*RightArm_h));


angle_BDF := angle_BDC + angle_CDE + DEG_TO_RAD(RightArm_angle_FDE);


angle_FDG := angle_BDF - (PI - theta2_rad);


points.x := -RightArm_w + RightArm_g*COS(theta2_rad) + RightArm_m*COS(angle_FDG);
points.y := RightArm_g*SIN(theta2_rad) + RightArm_m*SIN(angle_FDG);

RightArmFK := points;

END_FUNCTION

// ---- POUs/RightArmWristIK.TcPOU
FUNCTION RightArmWristIK : REAL
VAR_INPUT
	theta1:LREAL;			//右电机角度值
	theta2:LREAL;	        //左电机角度值
END_VAR                             
VAR                                 
	// 中间变量                         
	theta1_rad:LREAL;       //右电机弧度值
	theta2_rad:LREAL;       //左电机弧度值
	rr:LREAL;						//r变量被倍福占用了，所以此处用rr
	u:LREAL;
	angle_BDC:LREAL;
	angle_CDE:LREAL;
	angle_BDE:LREAL;
	angle_EDG:LREAL;

	
	point_E:Points;
	point_F:Points;
	
	jx:REAL;				//EF向量的横坐标
	jy:REAL;				//EF向量的纵坐标
	vx:REAL:=0;				//+y单位向量的横坐标
	vy:REAL:=1;				//+y单位向量的纵坐标
	result_cross:REAL;		//EF向量和+y向量的叉乘结果
	
	angle_Beta:REAL;
	
	
END_VAR

theta1_rad := DEG_TO_RAD(theta1);
theta2_rad := DEG_TO_RAD(theta2);

point_F := RightArmFK(theta1, theta2);

rr := SQRT(EXPT((2*RightArm_w+RightArm_f*COS(theta1_rad)-RightArm_g*COS(theta2_rad)),2) + EXPT((RightArm_f*SIN(theta1_rad)-RightArm_g*SIN(theta2_rad)),2));  

u := SQRT(EXPT((2*RightArm_w+RightArm_f*COS(theta1_rad)),2) + EXPT((RightArm_f*SIN(theta1_rad)),2));

angle_BDC := ACOS((rr*rr+RightArm_g*RightArm_g-u*u)/(2*rr*RightArm_g));

angle_CDE := ACOS((rr*rr + RightArm_h*RightArm_h -RightArm_i*RightArm_i)/(2*rr*RightArm_h));

angle_BDE := angle_BDC + angle_CDE;

angle_EDG := angle_BDE - (PI - theta2_rad);

point_E.x := -RightArm_w + RightArm_g*COS(theta2_rad) + RightArm_h*COS(angle_EDG);
point_E.y := RightArm_g*SIN(theta2_rad) + RightArm_h*SIN(angle_EDG);


jx := point_F.x - point_E.x;
jy := point_F.y - point_E.y;


result_cross := jx*vy - jy*vx;

IF result_cross > 0 THEN
	angle_Beta := ACOS((jx*vx+jy*vy)/(SQRT(jx*jx+jy*jy)*SQRT(vx*vx+vy*vy)));
ELSIF result_cross < 0 THEN
	angle_Beta := -ACOS((jx*vx+jy*vy)/(SQRT(jx*jx+jy*jy)*SQRT(vx*vx+vy*vy)));
ELSE
	angle_Beta := 0;
END_IF

RightArmWristIK := RAD_TO_DEG(angle_Beta);

END_FUNCTION

// ---- POUs/RightArmIK.TcPOU
FUNCTION RightArmIK : Angles
VAR_INPUT
	x:LREAL;
	y:LREAL;
END_VAR
VAR
	
	// 中间量
	p:LREAL;
	q:LREAL;
	k:LREAL;
	l:LREAL;
	angle_DBF:LREAL;	
	angle_OBF:LREAL;
	theta1:LREAL;
	theta2:LREAL;
	angle_BDF:LREAL;
	angle_BDE:LREAL;
	angle_DBE:LREAL;
	angle_EBA:LREAL;
	angle_EAB:LREAL;
	angle_CAE:LREAL;
	
	// 输出
	angles		:Angles;
	
END_VAR

// TWINCAT 角度换算以弧度为单位

p := SQRT((x+RightArm_w)*(x+RightArm_w)+y*y);
q := SQRT(x*x + y*y);
 
angle_DBF := ACOS((RightArm_g*RightArm_g+p*p-RightArm_m*RightArm_m)/(2*RightArm_g*p));
angle_OBF := ACOS((RightArm_w*RightArm_w+p*p-q*q)/(2*RightArm_w*p));
theta2 := angle_OBF + angle_DBF;

angle_BDF := ACOS((RightArm_g*RightArm_g+RightArm_m*RightArm_m-p*p)/(2*RightArm_g*RightArm_m));
//angle_FCE := ACOS((n*n+i*i-j*j)/(2*n*i));
angle_BDE := angle_BDF - DEG_TO_RAD(RightArm_angle_FDE);

k := SQRT(RightArm_h*RightArm_h+RightArm_g*RightArm_g-2*RightArm_h*RightArm_g*COS(angle_BDE));

angle_DBE := ACOS((RightArm_g*RightArm_g+k*k-RightArm_h*RightArm_h)/(2*RightArm_g*k));

angle_EBA := theta2 - angle_DBE;

l := SQRT(k*k + 4*RightArm_w*RightArm_w - 4*k*RightArm_w*COS(angle_EBA));

angle_EAB := ACOS((l*l+4*RightArm_w*RightArm_w-k*k)/(4*l*RightArm_w));

angle_CAE := ACOS((RightArm_f*RightArm_f+l*l-RightArm_i*RightArm_i)/(2*RightArm_f*l));

theta1 := PI - angle_CAE - angle_EAB;

angles.theta1_right := RAD_TO_DEG(theta1);
angles.theta2_left := RAD_TO_DEG(theta2);


RightArmIK := angles;

END_FUNCTION

// ---- POUs/RightArmManualCtrlMove.TcPOU
PROGRAM RightArmManualCtrlMove
VAR
	
	point												:Points;					// 当前腕关节坐标
	target_angle										:Angles;					// 臂左右电机目标角度
	manualState											:USINT;						// 手动控制状态标志位，0
	speed												:REAL := 0.5;					// 笛卡尔坐标位移速度
	x													:REAL;						// 腕关节目标位置x
	y													:REAL;						// 腕关节目标位置y
	wrist_angle											:REAL;						// 腕电机角度
	
	//左臂举升电机
	RightArm_Lift_Jog									:MC_Jog;
	bRightArm_Lift_Up									:BOOL;
	bRightArm_Lift_Down									:BOOL;
	nRightArmLiftSpeed									:LREAL:=3;
	
	
	RightArm_Right_ExtPosGen_Enable						:MC_ExtSetPointGenEnable;
	RightArm_Right_ExtPosGen_Disable                     :MC_ExtSetPointGenDisable;
	RightArm_Left_ExtPosGen_Enable                       :MC_ExtSetPointGenEnable;
	RightArm_Left_ExtPosGen_Disable	                    :MC_ExtSetPointGenDisable;
	RightArm_Wrist_ExtPosGen_Enable                      :MC_ExtSetPointGenEnable;
	RightArm_Wrist_ExtPosGen_Disable	                 :MC_ExtSetPointGenDisable;
	
	//串口
	//fb_SerialCom		:FB_SerialCom;					
	//wrist_angle_int		:INT;
	//wrist_angle_byte	:BYTE;
	
	
END_VAR

axis_RightArm_Left();
axis_RightArm_Right();
axis_RightArm_Wrist();
ExtPosGen();

// 外部位置发生器失能
RightArm_Right_ExtPosGen_Enable.Execute 		:= FALSE;
RightArm_Right_ExtPosGen_Disable.Execute 		:= FALSE;
RightArm_Left_ExtPosGen_Enable.Execute 			:= FALSE;
RightArm_Left_ExtPosGen_Disable.Execute 		:= FALSE;
RightArm_Wrist_ExtPosGen_Enable.Execute 		:= FALSE;
RightArm_Wrist_ExtPosGen_Disable.Execute 		:= FALSE;

IF bManualCtrl_Asm_RightArm THEN
	
	// 右臂举升电机Jog
	RightArmLiftJog();
	
	// 运动学正解出当前腕关节点坐标
	point := RightArmFK(axis_RightArm_Right.NcToPlc.ActPos, axis_RightArm_Left.NcToPlc.ActPos);
	
	// 用舵机进行程序验证的串口背景通讯
	//BackgroundSerialCtrl();
	
	IF bAutoCtrl_Part_RightWrist THEN
		
		wrist_angle := RightArmWristIK(axis_RightArm_Right.NcToPlc.ActPos, axis_RightArm_Left.NcToPlc.ActPos);		// 逆解出腕电机角度
		
	END_IF
	

	IF bRightArm_Forward THEN
		x := point.x;
		y := point.y + speed;
		target_angle := RightArmIK(x, y);
		manualState := 1;
		
	ELSIF bRightArm_Backward THEN
	
		x := point.x;
		y := point.y - speed;
		target_angle := RightArmIK(x, y);
		manualState := 1;
		
	ELSIF bRightArm_Left THEN
		
		x := point.x - speed;
		y := point.y;
		target_angle := RightArmIK(x, y);
		manualState := 1;
		
	ELSIF bRightArm_Right THEN
		
		x := point.x + speed;
		y := point.y;
		target_angle := RightArmIK(x, y);
		manualState := 1;
		
	ELSE
		manualState := 0;
	END_IF
	
	
	
	CASE manualState OF
		0:
			RightArm_Right_ExtPosGen_Enable.Execute 		:= FALSE;
			RightArm_Right_ExtPosGen_Disable.Execute 		:= TRUE;
			RightArm_Left_ExtPosGen_Enable.Execute 			:= FALSE;
			RightArm_Left_ExtPosGen_Disable.Execute 		:= TRUE;
			RightArm_Wrist_ExtPosGen_Enable.Execute 		:= FALSE;
			RightArm_Wrist_ExtPosGen_Disable.Execute 		:= TRUE;
		
		1:
			RightArm_Right_ExtPosGen_Enable.Execute 		:= TRUE;
			RightArm_Left_ExtPosGen_Enable.Execute 			:= TRUE;
			RightArm_Wrist_ExtPosGen_Enable.Execute 		:= TRUE;
			
			IF axis_RightArm_Right.Status.ExtSetPointGenEnabled AND axis_RightArm_Left.Status.ExtSetPointGenEnabled AND axis_RightArm_Wrist.Status.ExtSetPointGenEnabled THEN
				MC_ExtSetPointGenFeed(
					Position:= target_angle.theta1_right, 
					Velocity:= 5,  
					Acceleration:= 10,  
					Direction:= 1, 
					Axis:= axis_RightArm_Right);
		
				MC_ExtSetPointGenFeed(
					Position:= target_angle.theta2_left, 
					Velocity:= 5,  
					Acceleration:= 10,  
					Direction:= 1, 
					Axis:= axis_RightArm_Left);
					
				MC_ExtSetPointGenFeed(
					Position:= wrist_angle, 
					Velocity:= 5, 
					Acceleration:= 10, 
					Direction:= 1, 
					Axis:= axis_RightArm_Wrist);
			END_IF
	END_CASE

//ELSE

END_IF

ACTION ExtPosGen:
RightArm_Right_ExtPosGen_Enable(
	Axis:= axis_RightArm_Right, 
	Execute:= RightArm_Right_ExtPosGen_Enable.Execute, 
	Position:= , 
	PositionType:= , 
	Done=> , 
	Busy=> , 
	Error=> , 
	ErrorID=> , 
	Enabled=> );
	
RightArm_Right_ExtPosGen_Disable(
	Axis:= axis_RightArm_Right, 
	Execute:= RightArm_Right_ExtPosGen_Disable.Execute, 
	Done=> , 
	Busy=> , 
	Error=> , 
	ErrorID=> , 
	Enabled=> );
	
RightArm_Left_ExtPosGen_Enable(
	Axis:= axis_RightArm_Left, 
	Execute:= RightArm_Left_ExtPosGen_Enable.Execute, 
	Position:= , 
	PositionType:= , 
	Done=> , 
	Busy=> , 
	Error=> , 
	ErrorID=> , 
	Enabled=> );
	
RightArm_Left_ExtPosGen_Disable(
	Axis:= axis_RightArm_Left, 
	Execute:= RightArm_Left_ExtPosGen_Disable.Execute, 
	Done=> , 
	Busy=> , 
	Error=> , 
	ErrorID=> , 
	Enabled=> );
	
RightArm_Wrist_ExtPosGen_Enable(
	Axis:= axis_RightArm_Wrist, 
	Execute:= RightArm_Wrist_ExtPosGen_Enable.Execute, 
	Position:= , 
	PositionType:= , 
	Done=> , 
	Busy=> , 
	Error=> , 
	ErrorID=> , 
	Enabled=> );
	
RightArm_Wrist_ExtPosGen_Disable(
	Axis:= axis_RightArm_Wrist, 
	Execute:= RightArm_Wrist_ExtPosGen_Disable.Execute, 
	Done=> , 
	Busy=> , 
	Error=> , 
	ErrorID=> , 
	Enabled=> );
END_ACTION

ACTION RightArmLiftJog:
RightArm_Lift_Jog(
	Axis:= axis_RightArm_Lift, 
	JogForward:= bRightArm_Lift_Down, 
	JogBackwards:= bRightArm_Lift_Up, 
	Mode:= MC_JOGMODE_CONTINOUS, 
	Position:= , 
	Velocity:= nRightArmLiftSpeed, 
	Acceleration:= , 
	Deceleration:= , 
	Jerk:= , 
	Done=> , 
	Busy=> , 
	Active=> , 
	CommandAborted=> , 
	Error=> , 
	ErrorID=> );
END_ACTION

END_PROGRAM

// ---- POUs/WheelControl.TcPOU
PROGRAM WheelControl
VAR
	WheelDriver_ModesOfOperation		AT%Q* 	:SINT		:=8;			//手动关联到舵轮驱动器的RxPDO modes of operation标志位，PLC进入运行时将标志位置为8


	nWalkSpeed_Left								:LREAL		:=30;			//单位：mm/s
	nWalkSpeed_Right							:LREAL		:=30;			//单位：mm/s
	nSteerSpeed									:LREAL		:=5;			//单位：°/s
	nSteerSpeed_Moving							:LREAL		:=5;			//行进过程中转向速度
	
	axis_RightWheel_Steer_Manual_Jog			:Mc_Jog;
	nAxis_RightWheel_Steer_LimitAngle			:USINT		:=45;			// 舵机最大角度
	bAxis_RightWheel_Steer_AtLeftLimit			:BOOL;						// 右轮舵机到达左边界
	bAxis_RightWheel_Steer_AtRightLimit			:BOOL;						// 右轮舵机到达右边界
	nAxis_RightWheel_Steer_CurrentAngle			:INT;						// 右舵轮当前角度，为下面判断bAxis_RightWheel_Steer_NeedBackToOriginal而准备的，读取当前角度存储用的临时变量
	bAxis_RightWheel_Steer_NeedBackToOriginal	:BOOL;						// MotionType=7/8的情况下，也需要对右轮舵机的角度进行判断，如果超过nAxis_RightWheel_Steer_LimitAngle限制，则要进行回零操作，如果在限值范围内则直接开始运动
	
	MotionType									:USINT;						//大动作分类，0:待机状态；1：前进；2：后退，3：左平移，4：右平移, 5：左旋转，6，右旋转
	MotionStep									:USINT;						// 分动作，0：先转转向；1：再动行走电机
	
	fbRemoteCtrl_Up_Mode						:WheelCtrlButtonModeCheck;	// 判断上键按键模式：单击+hold/双击+hold
	fbRemoteCtrl_Down_Mode						:WheelCtrlButtonModeCheck;	// 判断下键按键模式：单击+hold/双击+hold
	fbRemoteCtrl_East_Mode						:WheelCtrlButtonModeCheck;	// 判断East键按键模式：单击+hold/双击+hold
	fbRemoteCtrl_West_Mode						:WheelCtrlButtonModeCheck;	// 判断West键按键模式：单击+hold/双击+hold
	fbRemoteCtrl_1Btn_Mode						:WheelCtrlButtonModeCheck;
	fbRemoteCtrl_2Btn_Mode						:WheelCtrlButtonModeCheck;
	
	
	LeftWheel_Walk_Direction					:MC_Direction;						// 前进标志位
	RightWheel_Walk_Direction					:MC_Direction;						// 前进标志位

	bPowerOn									:BOOL;								// 手动模式下，行走电机和转向电机上电。
	bChassisManualCtrl							:BOOL;								// 底盘手动模式
	bMoveFastMode								:BOOL;								// 底盘快速模式
	bMoveSlowMode								:BOOL		:=TRUE;					// 底盘慢速模式

	//test

	bAutoCtrl			:BOOL;
	
END_VAR

WheelPowerOn();	// 上电（目前是手动上电）
WheelWalkAxisMoveVelo();// 前进 or 后退
WheelSteerAxisMoveAbs();// 转向轴MoveAbs
WheelStop();

// 获取指定按键的点击模式	
fbRemoteCtrl_Up_Mode(bButton:= bRemoteCtrl_Up, bDoubleClickAndHold=> , bOnceClickAndHold=> );
fbRemoteCtrl_Down_Mode(bButton:= bRemoteCtrl_Down, bDoubleClickAndHold=> , bOnceClickAndHold=> );
fbRemoteCtrl_East_Mode(bButton:= bRemoteCtrl_East, bDoubleClickAndHold=> , bOnceClickAndHold=> );
fbRemoteCtrl_West_Mode(bButton:= bRemoteCtrl_West, bDoubleClickAndHold=> , bOnceClickAndHold=> );
fbRemoteCtrl_1Btn_Mode(bButton:= bRemoteCtrl_1Btn, bDoubleClickAndHold=> , bOnceClickAndHold=> );
fbRemoteCtrl_2Btn_Mode(bButton:= bRemoteCtrl_2Btn, bDoubleClickAndHold=> , bOnceClickAndHold=> );


// 手动模式激活后此标志位置true，转向和行走电机上电
bPowerOn := FALSE;


// 底盘手动模式标志位
bChassisManualCtrl := FALSE;


//当手动遥控Online置位且舵轮上电
IF bRemoteCtrl_Online THEN
	
	// 上电
	bPowerOn := TRUE;
	
	// 底盘手动模式标志位
	bChassisManualCtrl := TRUE;
	
	// 手动调整右轮舵机角度，里面有按键互斥以及到达限位的逻辑
	RightWheelSteerJog();
	
	// 按键都没按下，待机模式
	IF NOT bRemoteCtrl_Up AND NOT bRemoteCtrl_Down AND NOT bRemoteCtrl_East AND NOT bRemoteCtrl_West AND NOT bRemoteCtrl_South AND NOT bRemoteCtrl_North AND NOT bRemoteCtrl_1btn AND NOT bRemoteCtrl_2btn THEN
		MotionType 		:= 0;
		MotionStep		:=0;
	END_IF
	

	//MotionType:=1-6时，手动调整右轮舵机的Mc_Jog,判断逻辑再RightWheelSteerJog中
	// 长按遥控器“上”键，车先把舵转向0度，再前进
	IF fbRemoteCtrl_Up_Mode.bOnceClickAndHold THEN
		
		MotionType := 1;
		
	END_IF
	
	// 长按遥控器“下”, 车先把舵转向0度，再后退
	IF fbRemoteCtrl_Down_Mode.bOnceClickAndHold THEN
		
		MotionType := 2;
		
	END_IF
	
	// 长按遥控器“东”,车先把舵转向90度， 车左平移
	IF fbRemoteCtrl_East_Mode.bOnceClickAndHold THEN
		
		MotionType := 3;
		
	END_IF
	
	// 长按遥控器“西”,车先把舵转向90度， 车右平移
	IF fbRemoteCtrl_West_Mode.bOnceClickAndHold THEN
		
		MotionType := 4;
		
	END_IF
	
	// 双击+长按遥控器“东”,车先把舵转向54.0903度， 车左旋转
	IF fbRemoteCtrl_East_Mode.bDoubleClickAndHold THEN
		
		MotionType := 5;
		
	END_IF
	
	// 双击+长按遥控器“西”,车先把舵转向54.0903度，, 车右旋转
	IF fbRemoteCtrl_West_Mode.bDoubleClickAndHold THEN
		
		MotionType := 6;
		
	END_IF
	
	// 双击+长按遥控器“up”,车以当前舵机角度前进，行进中可以调整舵机
	IF fbRemoteCtrl_Up_Mode.bDoubleClickAndHold THEN
		
		MotionType := 7;
		
	END_IF
	
	// 双击+长按遥控器“down”,车以当前舵机角度后退，行进中可以调整舵机
	IF fbRemoteCtrl_Down_Mode.bDoubleClickAndHold THEN
		
		MotionType := 8;
		
	END_IF
	
	
	// 单击+长按 button_1，激活慢速模式（默认）
	IF fbRemoteCtrl_1Btn_Mode.bOnceClickAndHold THEN
	
		bMoveSlowMode 							:= TRUE;
		bMoveFastMode 							:= FALSE;
		nWalkSpeed_Left							:=30;			//单位：mm/s
		nWalkSpeed_Right						:=30;			//单位：mm/s
		nSteerSpeed								:=5;			//单位：°/s
		nSteerSpeed_Moving						:=5;			//行进过程中转向速度
	END_IF
	
	// 单击+长按 button_2，激活快速模式
	IF fbRemoteCtrl_2Btn_Mode.bOnceClickAndHold THEN
	
		bMoveSlowMode 							:= FALSE ;
		bMoveFastMode 							:= TRUE;
		nWalkSpeed_Left							:=60;			//单位：mm/s
		nWalkSpeed_Right						:=60;			//单位：mm/s
		nSteerSpeed								:=10;			//单位：°/s
		nSteerSpeed_Moving						:=10;			//行进过程中转向速度
		
	END_IF
	
END_IF


CASE MotionType OF
	
	// 激活底盘遥控时待机状态
	0:

		
		MotionStep		:=0;
		
		
		axis_LeftWheel_Steer_MoveAbs.Execute := FALSE;
		axis_RightWheel_Steer_MoveAbs.Execute := FALSE;
		
		axis_LeftWheel_Walk_MoveVelo.Execute := FALSE;
		axis_RightWheel_Walk_MoveVelo.Execute := FALSE;
		

		axis_RightWheel_Steer_McStop(Axis:= axis_RightWheel_Steer, Execute:= FALSE);
		axis_RightWheel_Walk_McStop(Axis:= axis_RightWheel_Walk, Execute:= FALSE);
		axis_LeftWheel_Steer_McStop(Axis:= axis_LeftWheel_Steer, Execute:= FALSE);
		axis_LeftWheel_Walk_McStop(Axis:= axis_LeftWheel_Walk, Execute:= FALSE);
		
		
		
		IF axis_LeftWheel_Steer_MoveAbs.Active OR axis_RightWheel_Steer_MoveAbs.Active OR axis_LeftWheel_Walk_MoveVelo.Active OR axis_RightWheel_Walk_MoveVelo.Active THEN

			axis_RightWheel_Steer_McStop(Axis:= axis_RightWheel_Steer, Execute:= TRUE);
			axis_RightWheel_Walk_McStop(Axis:= axis_RightWheel_Walk, Execute:= TRUE);
			axis_LeftWheel_Steer_McStop(Axis:= axis_LeftWheel_Steer, Execute:= TRUE);
			axis_LeftWheel_Walk_McStop(Axis:= axis_LeftWheel_Walk, Execute:= TRUE);
		END_IF 

		
		
	// 前进
	1:
		CASE MotionStep OF
			
			// 控制舵机旋转到零
			0:
				axis_LeftWheel_Steer_MoveAbs.Position := 0;
				axis_RightWheel_Steer_MoveAbs.Position := 0;
				axis_LeftWheel_Steer_MoveAbs.Velocity := nSteerSpeed;
				axis_RightWheel_Steer_MoveAbs.Velocity := nSteerSpeed;				
				axis_LeftWheel_Steer_MoveAbs.Execute := TRUE;
				axis_RightWheel_Steer_MoveAbs.Execute := TRUE;
				
				
				
				IF axis_LeftWheel_Steer_MoveAbs.Done = TRUE AND axis_RightWheel_Steer_MoveAbs.Done = TRUE THEN
					axis_LeftWheel_Steer_MoveAbs.Execute := FALSE;
					axis_RightWheel_Steer_MoveAbs.Execute := FALSE;
					MotionStep := 1;
				END_IF
			1:
				axis_LeftWheel_Walk_MoveVelo.Direction := MC_Positive_Direction;
				axis_RightWheel_Walk_MoveVelo.Direction := MC_Negative_Direction;
				axis_LeftWheel_Walk_MoveVelo.Execute := TRUE;
				axis_RightWheel_Walk_MoveVelo.Execute := TRUE;				

		END_CASE

		
	// 后退
	2:
		CASE MotionStep OF
		
			// 控制舵机旋转到零
			0:
				axis_LeftWheel_Steer_MoveAbs.Position := 0;
				axis_RightWheel_Steer_MoveAbs.Position := 0;
				axis_LeftWheel_Steer_MoveAbs.Velocity := nSteerSpeed;
				axis_RightWheel_Steer_MoveAbs.Velocity := nSteerSpeed;				
				axis_LeftWheel_Steer_MoveAbs.Execute := TRUE;
				axis_RightWheel_Steer_MoveAbs.Execute := TRUE;
				
				IF axis_LeftWheel_Steer_MoveAbs.Done = TRUE AND axis_RightWheel_Steer_MoveAbs.Done = TRUE THEN
					axis_LeftWheel_Steer_MoveAbs.Execute := FALSE;
					axis_RightWheel_Steer_MoveAbs.Execute := FALSE;
					MotionStep := 1;
				END_IF
			1:
				axis_LeftWheel_Walk_MoveVelo.Direction := MC_Negative_Direction;
				axis_RightWheel_Walk_MoveVelo.Direction := MC_Positive_Direction;
				axis_LeftWheel_Walk_MoveVelo.Execute := TRUE;
				axis_RightWheel_Walk_MoveVelo.Execute := TRUE;				
											  
											  
		END_CASE
	
	// 向右平移	
	3:
		CASE MotionStep OF
		
			// 控制舵机旋转到90度
			0:
				axis_LeftWheel_Steer_MoveAbs.Position := 90;
				axis_RightWheel_Steer_MoveAbs.Position := 90;
				axis_LeftWheel_Steer_MoveAbs.Velocity := nSteerSpeed;
				axis_RightWheel_Steer_MoveAbs.Velocity := nSteerSpeed;				
				axis_LeftWheel_Steer_MoveAbs.Execute := TRUE;
				axis_RightWheel_Steer_MoveAbs.Execute := TRUE;
				
				IF axis_LeftWheel_Steer_MoveAbs.Done = TRUE AND axis_RightWheel_Steer_MoveAbs.Done = TRUE THEN
					axis_LeftWheel_Steer_MoveAbs.Execute := FALSE;
					axis_RightWheel_Steer_MoveAbs.Execute := FALSE;
					MotionStep := 1;
				END_IF
			1:
				axis_LeftWheel_Walk_MoveVelo.Direction := MC_Negative_Direction;
				axis_RightWheel_Walk_MoveVelo.Direction := MC_Positive_Direction;
				axis_LeftWheel_Walk_MoveVelo.Execute := TRUE;
				axis_RightWheel_Walk_MoveVelo.Execute := TRUE;			
		END_CASE
		
		
	// 向左平移	
	4:
		CASE MotionStep OF
		
			// 控制舵机旋转到90度
			0:
				axis_LeftWheel_Steer_MoveAbs.Position := 90;
				axis_RightWheel_Steer_MoveAbs.Position := 90;
				axis_LeftWheel_Steer_MoveAbs.Velocity := nSteerSpeed;
				axis_RightWheel_Steer_MoveAbs.Velocity := nSteerSpeed;				
				axis_LeftWheel_Steer_MoveAbs.Execute := TRUE;
				axis_RightWheel_Steer_MoveAbs.Execute := TRUE;
				
				IF axis_LeftWheel_Steer_MoveAbs.Done = TRUE AND axis_RightWheel_Steer_MoveAbs.Done = TRUE THEN
					axis_LeftWheel_Steer_MoveAbs.Execute := FALSE;
					axis_RightWheel_Steer_MoveAbs.Execute := FALSE;
					MotionStep := 1;
				END_IF
			1:
				axis_LeftWheel_Walk_MoveVelo.Direction := MC_Positive_Direction;
				axis_RightWheel_Walk_MoveVelo.Direction := MC_Negative_Direction;
				axis_LeftWheel_Walk_MoveVelo.Execute := TRUE;
				axis_RightWheel_Walk_MoveVelo.Execute := TRUE;			
		END_CASE
	
		
	// 原地向左旋转	
	5:
		CASE MotionStep OF
		
			// 控制舵机旋转到54.0903度
			0:
				axis_LeftWheel_Steer_MoveAbs.Position := 54.0903;
				axis_RightWheel_Steer_MoveAbs.Position := 54.0903;
				axis_LeftWheel_Steer_MoveAbs.Velocity := nSteerSpeed;
				axis_RightWheel_Steer_MoveAbs.Velocity := nSteerSpeed;				
				axis_LeftWheel_Steer_MoveAbs.Execute := TRUE;
				axis_RightWheel_Steer_MoveAbs.Execute := TRUE;
				
				IF axis_LeftWheel_Steer_MoveAbs.Done = TRUE AND axis_RightWheel_Steer_MoveAbs.Done = TRUE THEN
					axis_LeftWheel_Steer_MoveAbs.Execute := FALSE;
					axis_RightWheel_Steer_MoveAbs.Execute := FALSE;
					MotionStep := 1;
				END_IF
			1:
				axis_LeftWheel_Walk_MoveVelo.Direction := MC_Negative_Direction;
				axis_RightWheel_Walk_MoveVelo.Direction := MC_Negative_Direction;
				axis_LeftWheel_Walk_MoveVelo.Execute := TRUE;
				axis_RightWheel_Walk_MoveVelo.Execute := TRUE;
			
		END_CASE
		
		
	// 原地向右旋转	
	6:
		CASE MotionStep OF
		
			// 控制舵机旋转到54.0903度
			0:
				axis_LeftWheel_Steer_MoveAbs.Position := 54.0903;
				axis_RightWheel_Steer_MoveAbs.Position := 54.0903;
				axis_LeftWheel_Steer_MoveAbs.Velocity := nSteerSpeed;
				axis_RightWheel_Steer_MoveAbs.Velocity := nSteerSpeed;				
				axis_LeftWheel_Steer_MoveAbs.Execute := TRUE;
				axis_RightWheel_Steer_MoveAbs.Execute := TRUE;
				
				IF axis_LeftWheel_Steer_MoveAbs.Done = TRUE AND axis_RightWheel_Steer_MoveAbs.Done = TRUE THEN
					axis_LeftWheel_Steer_MoveAbs.Execute := FALSE;
					axis_RightWheel_Steer_MoveAbs.Execute := FALSE;
					MotionStep := 1;
				END_IF
			1:
				axis_LeftWheel_Walk_MoveVelo.Direction := MC_Positive_Direction;
				axis_RightWheel_Walk_MoveVelo.Direction := MC_Positive_Direction;
				axis_LeftWheel_Walk_MoveVelo.Execute := TRUE;
				axis_RightWheel_Walk_MoveVelo.Execute := TRUE;
			
		END_CASE
		

	// 前进中调整舵机
	7:
	
		CASE MotionStep OF
			
			//先判断右舵机是否需要归零位
			0:
				nAxis_RightWheel_Steer_CurrentAngle := (TO_INT(axis_RightWheel_Steer.NcToPlc.ActPos*100)/100);	// 读取右舵轮当前角度，判断是否超限制，超限值需要归0位
				
				//MotionType=7/8的情况下，也需要对右轮舵机的角度进行判断，如果超过nAxis_RightWheel_Steer_LimitAngle限制，则右舵机要进行回零操作，如果在限值范围内则直接开始运f动
				IF nAxis_RightWheel_Steer_CurrentAngle >= nAxis_RightWheel_Steer_LimitAngle OR nAxis_RightWheel_Steer_CurrentAngle <= -nAxis_RightWheel_Steer_LimitAngle THEN
					bAxis_RightWheel_Steer_NeedBackToOriginal := TRUE;
				ELSE
					bAxis_RightWheel_Steer_NeedBackToOriginal := FALSE;
				END_IF
				
				MotionStep := 1;
			
			//把左前舵机和右后舵机（视情况）旋转置0位
			1:	
				// 左舵机置零位
				axis_LeftWheel_Steer_MoveAbs.Position := 0;
				axis_LeftWheel_Steer_MoveAbs.Velocity := nSteerSpeed;
				axis_LeftWheel_Steer_MoveAbs.Execute := TRUE;

				// 如果右舵轮需要回0
				IF bAxis_RightWheel_Steer_NeedBackToOriginal THEN
					axis_RightWheel_Steer_MoveAbs.Position := 0;
					axis_RightWheel_Steer_MoveAbs.Velocity := nSteerSpeed;
					axis_RightWheel_Steer_MoveAbs.Execute := TRUE;
					
					IF axis_LeftWheel_Steer_MoveAbs.Done = TRUE AND axis_RightWheel_Steer_MoveAbs.Done = TRUE THEN
						axis_LeftWheel_Steer_MoveAbs.Execute := FALSE;
						axis_RightWheel_Steer_MoveAbs.Execute := FALSE;
						bAxis_RightWheel_Steer_NeedBackToOriginal := FALSE;
						MotionStep := 2;
					END_IF
				ELSE	// 仅需左前舵机归0
					IF axis_LeftWheel_Steer_MoveAbs.Done = TRUE THEN
						axis_LeftWheel_Steer_MoveAbs.Execute := FALSE;
						MotionStep := 2;
					END_IF
				END_IF


			//左右轮差速运动，左轮速度为基准，右轮根据右舵的角度实时差速
			2:
				// 若要实时更新Mc_MoveVelocity的速度值，需要重新触发一次，Excecute先置False
				axis_RightWheel_Walk_MoveVelo(Axis:= axis_RightWheel_Walk, 	Execute:= FALSE);
				
				// 根据舵机角度实时计算行走电机速度
				nWalkSpeed_Right := WheelWalkDifferential(TO_INT(axis_RightWheel_Steer.NcToPlc.ActPos*100)/100);	// 保留两位小数
				
				// 设置行走电机方向
				axis_LeftWheel_Walk_MoveVelo.Direction := MC_Positive_Direction;
				axis_RightWheel_Walk_MoveVelo.Direction := MC_Negative_Direction;
				
				// 设置左右行走电机速度
				axis_LeftWheel_Walk_MoveVelo.Velocity := nWalkSpeed_Left;
				axis_RightWheel_Walk_MoveVelo.Velocity := nWalkSpeed_Right;
				
				axis_LeftWheel_Walk_MoveVelo.Execute := TRUE;
				axis_RightWheel_Walk_MoveVelo.Execute := TRUE;
				
		END_CASE
		

	
		
	// 后退中调整舵机
	8:
	
		CASE MotionStep OF
			
//			//先把左前舵机旋转置0位
//			0:
//				axis_LeftWheel_Steer_MoveAbs.Position := 0;
//				axis_LeftWheel_Steer_MoveAbs.Velocity := 5;				
//				axis_LeftWheel_Steer_MoveAbs.Execute := TRUE;

//				IF axis_LeftWheel_Steer_MoveAbs.Done = TRUE THEN
					
//					axis_LeftWheel_Steer_MoveAbs.Execute := FALSE;
//					MotionStep := 1;
//				END_IF
			
//			//左右轮差速运动，左轮速度为基准，右轮根据右舵的角度实时差速
//			1:
			
//				// 需要再触发实现速度实时更新
//				axis_RightWheel_Walk_MoveVelo(Axis:= axis_RightWheel_Walk, 	Execute:= FALSE);
				
//				// 根据舵机角度实时计算行走电机速度
//				nWalkSpeed_Right := WheelWalkDifferential(TO_INT(axis_RightWheel_Steer.NcToPlc.ActPos*100)/100);	// 保留两位小数
				
//				// 设置行走电机方向
//				axis_LeftWheel_Walk_MoveVelo.Direction := MC_Negative_Direction;
//				axis_RightWheel_Walk_MoveVelo.Direction := MC_Positive_Direction;
				
//				// 设置左右行走电机速度
//				axis_LeftWheel_Walk_MoveVelo.Velocity := nWalkSpeed_Left;
//				axis_RightWheel_Walk_MoveVelo.Velocity := nWalkSpeed_Right;
				
//				// 再次触发
//				axis_LeftWheel_Walk_MoveVelo.Execute := TRUE;
//				axis_RightWheel_Walk_MoveVelo.Execute := TRUE;	

			//先判断右舵机是否需要归零位
			0:
				nAxis_RightWheel_Steer_CurrentAngle := (TO_INT(axis_RightWheel_Steer.NcToPlc.ActPos*100)/100);	// 读取右舵轮当前角度，判断是否超限制，超限值需要归0位
				
				//MotionType=7/8的情况下，也需要对右轮舵机的角度进行判断，如果超过nAxis_RightWheel_Steer_LimitAngle限制，则右舵机要进行回零操作，如果在限值范围内则直接开始运f动
				IF nAxis_RightWheel_Steer_CurrentAngle >= nAxis_RightWheel_Steer_LimitAngle OR nAxis_RightWheel_Steer_CurrentAngle <= -nAxis_RightWheel_Steer_LimitAngle THEN
					bAxis_RightWheel_Steer_NeedBackToOriginal := TRUE;
				ELSE
					bAxis_RightWheel_Steer_NeedBackToOriginal := FALSE;
				END_IF
				
				MotionStep := 1;
			
			//把左前舵机和右后舵机（视情况）旋转置0位
			1:	
				// 左舵机置零位
				axis_LeftWheel_Steer_MoveAbs.Position := 0;
				axis_LeftWheel_Steer_MoveAbs.Velocity := nSteerSpeed;
				axis_LeftWheel_Steer_MoveAbs.Execute := TRUE;

				// 如果右舵轮需要回0
				IF bAxis_RightWheel_Steer_NeedBackToOriginal THEN
					axis_RightWheel_Steer_MoveAbs.Position := 0;
					axis_RightWheel_Steer_MoveAbs.Velocity := nSteerSpeed;
					axis_RightWheel_Steer_MoveAbs.Execute := TRUE;
					
					IF axis_LeftWheel_Steer_MoveAbs.Done = TRUE AND axis_RightWheel_Steer_MoveAbs.Done = TRUE THEN
						axis_LeftWheel_Steer_MoveAbs.Execute := FALSE;
						axis_RightWheel_Steer_MoveAbs.Execute := FALSE;
						bAxis_RightWheel_Steer_NeedBackToOriginal := FALSE;
						MotionStep := 2;
					END_IF
				ELSE	// 仅需左前舵机归0
					IF axis_LeftWheel_Steer_MoveAbs.Done = TRUE THEN
						axis_LeftWheel_Steer_MoveAbs.Execute := FALSE;
						MotionStep := 2;
					END_IF
				END_IF


			//左右轮差速运动，左轮速度为基准，右轮根据右舵的角度实时差速
			2:
				// 若要实时更新Mc_MoveVelocity的速度值，需要重新触发一次，Excecute先置False
				axis_RightWheel_Walk_MoveVelo(Axis:= axis_RightWheel_Walk, 	Execute:= FALSE);
				
				// 根据舵机角度实时计算行走电机速度
				nWalkSpeed_Right := WheelWalkDifferential(TO_INT(axis_RightWheel_Steer.NcToPlc.ActPos*100)/100);	// 保留两位小数
				
				// 设置行走电机方向
				axis_LeftWheel_Walk_MoveVelo.Direction := MC_Negative_Direction; 
				axis_RightWheel_Walk_MoveVelo.Direction := MC_Positive_Direction;
				
				// 设置左右行走电机速度
				axis_LeftWheel_Walk_MoveVelo.Velocity := nWalkSpeed_Left;
				axis_RightWheel_Walk_MoveVelo.Velocity := nWalkSpeed_Right;
				
				axis_LeftWheel_Walk_MoveVelo.Execute := TRUE;
				axis_RightWheel_Walk_MoveVelo.Execute := TRUE;
		
		END_CASE
		
END_CASE

	

// 自动
//IF bAutoCtrl AND bPowerOn THEN
	
//END_IF

ACTION RightWheelSteerJog:
// 到达极限位置后标志位置true，不再Jog，只能向相反的方向jog
IF axis_RightWheel_Steer.NcToPlc.ActPos >= nAxis_RightWheel_Steer_LimitAngle THEN
	bAxis_RightWheel_Steer_AtRightLimit := TRUE;										// 右轮舵机>=nAxis_RightWheel_Steer_LimitAngle度时，视为到达右边界，bAxis_RightWheel_Steer_AtRightLimit置位，下方的判断会造成舵机不再右转
ELSIF axis_RightWheel_Steer.NcToPlc.ActPos <= -nAxis_RightWheel_Steer_LimitAngle THEN
	bAxis_RightWheel_Steer_AtLeftLimit := TRUE;											// 右轮舵机<=-nAxis_RightWheel_Steer_LimitAngle度时，视为到达左边界,同上
ELSE
	bAxis_RightWheel_Steer_AtRightLimit := FALSE;
	bAxis_RightWheel_Steer_AtLeftLimit := FALSE;
END_IF

axis_RightWheel_Steer_Manual_Jog(
	Axis:= axis_RightWheel_Steer, 
	JogForward:= bRemoteCtrl_South AND NOT bAxis_RightWheel_Steer_AtRightLimit AND NOT fbRemoteCtrl_Up_Mode.bOnceClickAndHold AND NOT fbRemoteCtrl_Down_Mode.bOnceClickAndHold AND NOT fbRemoteCtrl_East_Mode.bOnceClickAndHold AND NOT fbRemoteCtrl_West_Mode.bOnceClickAndHold AND NOT fbRemoteCtrl_East_Mode.bDoubleClickAndHold AND NOT fbRemoteCtrl_West_Mode.bDoubleClickAndHold, 
	JogBackwards:= bRemoteCtrl_North AND NOT bAxis_RightWheel_Steer_AtLeftLimit AND NOT fbRemoteCtrl_Up_Mode.bOnceClickAndHold AND NOT fbRemoteCtrl_Down_Mode.bOnceClickAndHold AND NOT fbRemoteCtrl_East_Mode.bOnceClickAndHold AND NOT fbRemoteCtrl_West_Mode.bOnceClickAndHold AND NOT fbRemoteCtrl_East_Mode.bDoubleClickAndHold AND NOT fbRemoteCtrl_West_Mode.bDoubleClickAndHold, 
	Mode:= MC_JOGMODE_CONTINOUS, 
	Position:= , 
	Velocity:= nSteerSpeed_Moving, 
	Acceleration:= , 
	Deceleration:= , 
	Jerk:= , 
	Done=> , 
	Busy=> , 
	Active=> , 
	CommandAborted=> , 
	Error=> , 
	ErrorID=> );
END_ACTION

ACTION WheelPowerOn:
axis_RightWheel_Walk_Power(
	Axis:= axis_RightWheel_Walk, 
	Enable:= bPowerOn, 
	Enable_Positive:= TRUE, 
	Enable_Negative:= TRUE, 
	Override:= , 
	BufferMode:= , 
	Options:= , 
	Status=> , 
	Busy=> , 
	Error=> , 
	ErrorID=> );
	
axis_LeftWheel_Walk_Power(
	Axis:= axis_LeftWheel_Walk, 
	Enable:= bPowerOn, 
	Enable_Positive:= TRUE, 
	Enable_Negative:= TRUE, 
	Override:= , 
	BufferMode:= , 
	Options:= , 
	Status=> , 
	Busy=> , 
	Error=> , 
	ErrorID=> );

axis_RightWheel_Steer_Power(
	Axis:= axis_RightWheel_Steer, 
	Enable:= bPowerOn, 
	Enable_Positive:= TRUE, 
	Enable_Negative:= TRUE, 
	Override:= , 
	BufferMode:= , 
	Options:= , 
	Status=> , 
	Busy=> , 
	Error=> , 
	ErrorID=> );
	
axis_LeftWheel_Steer_Power(
	Axis:= axis_LeftWheel_Steer, 
	Enable:= bPowerOn, 
	Enable_Positive:= TRUE, 
	Enable_Negative:= TRUE, 
	Override:= , 
	BufferMode:= , 
	Options:= , 
	Status=> , 
	Busy=> , 
	Error=> , 
	ErrorID=> );
END_ACTION

ACTION WheelSteerAxisMoveAbs:
axis_LeftWheel_Steer_MoveAbs(
	Axis:= axis_LeftWheel_Steer, 
	Execute:= axis_LeftWheel_Steer_MoveAbs.Execute, 
	Position:= axis_LeftWheel_Steer_MoveAbs.Position, 
	Velocity:= axis_LeftWheel_Steer_MoveAbs.Velocity, 
	Acceleration:= , 
	Deceleration:= , 
	Jerk:= , 
	BufferMode:= , 
	Options:= , 
	Done=> , 
	Busy=> , 
	Active=> , 
	CommandAborted=> , 
	Error=> , 
	ErrorID=> );
	
	
axis_RightWheel_Steer_MoveAbs(
	Axis:= axis_RightWheel_Steer, 
	Execute:= axis_RightWheel_Steer_MoveAbs.Execute, 
	Position:= axis_RightWheel_Steer_MoveAbs.Position, 
	Velocity:= axis_RightWheel_Steer_MoveAbs.Velocity, 
	Acceleration:= , 
	Deceleration:= , 
	Jerk:= , 
	BufferMode:= , 
	Options:= , 
	Done=> , 
	Busy=> , 
	Active=> , 
	CommandAborted=> , 
	Error=> , 
	ErrorID=> );
END_ACTION

ACTION WheelStop:
axis_LeftWheel_Steer_McStop(
	Axis:= axis_LeftWheel_Steer, 
	Execute:= axis_LeftWheel_Steer_McStop.Execute, 
	Deceleration:= , 
	Jerk:= , 
	Options:= , 
	Done=> , 
	Busy=> , 
	Active=> , 
	CommandAborted=> , 
	Error=> , 
	ErrorID=> );
	
axis_LeftWheel_Walk_McStop(
	Axis:= axis_LeftWheel_Walk, 
	Execute:= axis_LeftWheel_Walk_McStop.Execute, 
	Deceleration:= , 
	Jerk:= , 
	Options:= , 
	Done=> , 
	Busy=> , 
	Active=> , 
	CommandAborted=> , 
	Error=> , 
	ErrorID=> );
	
axis_RightWheel_Steer_McStop(
	Axis:= axis_RightWheel_Steer, 
	Execute:= axis_RightWheel_Steer_McStop.Execute, 
	Deceleration:= , 
	Jerk:= , 
	Options:= , 
	Done=> , 
	Busy=> , 
	Active=> , 
	CommandAborted=> , 
	Error=> , 
	ErrorID=> );
	
axis_RightWheel_Walk_McStop(
	Axis:= axis_RightWheel_Walk, 
	Execute:= axis_RightWheel_Walk_McStop.Execute, 
	Deceleration:= , 
	Jerk:= , 
	Options:= , 
	Done=> , 
	Busy=> , 
	Active=> , 
	CommandAborted=> , 
	Error=> , 
	ErrorID=> );
END_ACTION

ACTION WheelWalkAxisMoveVelo:
axis_RightWheel_Walk_MoveVelo(
	Axis:= axis_RightWheel_Walk, 
	Execute:= axis_RightWheel_Walk_MoveVelo.Execute, 
	Velocity:= nWalkSpeed_Right, 
	Acceleration:= , 
	Deceleration:= , 
	Jerk:= , 
	Direction:= axis_RightWheel_Walk_MoveVelo.Direction, 
	BufferMode:= , 
	Options:= , 
	InVelocity=> , 
	Busy=> , 
	Active=> , 
	CommandAborted=> , 
	Error=> , 
	ErrorID=> );
	
axis_LeftWheel_Walk_MoveVelo(
	Axis:= axis_LeftWheel_Walk, 
	Execute:= axis_LeftWheel_Walk_MoveVelo.Execute, 
	Velocity:= nWalkSpeed_Left, 
	Acceleration:= , 
	Deceleration:= , 
	Jerk:= , 
	Direction:= axis_LeftWheel_Walk_MoveVelo.Direction, 
	BufferMode:= , 
	Options:= , 
	InVelocity=> , 
	Busy=> , 
	Active=> , 
	CommandAborted=> , 
	Error=> , 
	ErrorID=> );
END_ACTION

METHOD WheelWalkDifferential : LREAL
VAR_INPUT
	RightWheelSteerAngle		: LREAL;		// 右后轮转向角，正值轮右转，车左转；负值轮左转，车右转
END_VAR

VAR
	LK							: LREAL:=1450;					// 前后轴距1450
	LJ							: LREAL:=1050;
	RightWheelSteerAngle_RAD	: LREAL;						// 转向角弧度值			
	v_HG						: LREAL;						// 右后轮线速度
	v_AB						: LREAL :=nWalkSpeed_Left;		// 左前轮线速度
	R_KI						: LREAL;						// 右轮转弯半径
	R_JI						: LREAL;						// 左轮转弯半径
END_VAR
RightWheelSteerAngle_RAD := DEG_TO_RAD(RightWheelSteerAngle);

IF RightWheelSteerAngle = 0 THEN
	R_KI:=1;
	R_JI:=1;
ELSIF RightWheelSteerAngle > 0 THEN
	R_JI := LK/(TAN(RightWheelSteerAngle_RAD)) - LJ;
	R_KI := LK/SIN(RightWheelSteerAngle_RAD);
ELSIF RightWheelSteerAngle < 0 THEN
	R_JI := LK/(TAN(-RightWheelSteerAngle_RAD)) + LJ;
	R_KI := LK/SIN(-RightWheelSteerAngle_RAD);
END_IF

v_HG := (R_KI/R_JI)*v_AB;

WheelWalkDifferential := v_HG;
END_METHOD

END_PROGRAM

// ---- POUs/WheelCtrlButtonModeCheck.TcPOU
FUNCTION_BLOCK WheelCtrlButtonModeCheck
VAR_INPUT
	bButton		: BOOL;
	
END_VAR
VAR_OUTPUT
	
	bDoubleClickAndHold			:BOOL;										// true: double click and hold
	bOnceClickAndHold			:BOOL;										// true: once click and hold

END_VAR
VAR
	tonClickTimer								:TON;						// 点击计时器，tDoubleClickTime时间内点击点击两次为双击，超时则为单机
	tDoubleClickTime							:TIME	:=T#2000MS;			// 2000ms内认为是双击
	
	tonHoldTimer								:TON;						// 双击hold计时器，双击后hold住开始计时，超过tHoldTime则视为双击+Hold
	tHoldTime									:TIME	:=T#2000MS;			// 
	
	cClickCnt									:CTU;						// 点击次数计数器,2次触发reset信号


	
	bHold					:BOOL;
	nStep					:USINT;

END_VAR

(*
功能说明：

1、当检测到按键点击时，进入nstep=1，开启tonClickTimer定时器，进行按键模式检测；

2、在定时器触发ON之前，如果再点击按钮，则视为检测到双击，进入nStep=2，进入nstep2后开始检测按键是否双击后hold，如果hold，则bDoubleClickAndHold置true，如果送开则回nstep=0；

3、如果在tonClickTimer定时器触发ON前松手,则返回nSteop=0;如果在tonClickTimer定时器触发ON之后还检测到BUTTON一直被按下，则进入nStep=3，单击+hold模式，如果松开则回到nstep=0待机模式。
*)


